gfCNCPoint4[14464] = {X 340.3975, Y 90.3624, Z -5.5000, A 0.000, B 0.000, C 0.000 }
gfCNCPoint4[14465] = {X 344.7798, Y 90.5164, Z -5.5000, A 0.000, B 0.000, C 0.000 }
gfCNCPoint4[14466] = {X 349.1649, Y 90.5297, Z -5.5000, A 0.000, B 0.000, C 0.000 }
gfCNCPoint4[14467] = {X 353.3215, Y 90.4612, Z -5.5000, A 0.000, B 0.000, C 0.000 }
gfCNCPoint4[14468] = {X 357.4730, Y 90.2419, Z -5.5000, A 0.000, B 0.000, C 0.000 }
gfCNCPoint4[14469] = {X 361.6137, Y 89.8721, Z -5.5000, A 0.000, B 0.000, C 0.000 }
gfCNCPoint4[14470] = {X 363.7037, Y 89.5838, Z -5.5000, A 0.000, B 0.000, C 0.000 }
gfCNCPoint4[14471] = {X 365.7746, Y 89.1801, Z -5.5000, A 0.000, B 0.000, C 0.000 }
gfCNCPoint4[14472] = {X 367.8199, Y 88.6622, Z -5.5000, A 0.000, B 0.000, C 0.000 }
gfCNCPoint4[14473] = {X 368.7685, Y 88.3433, Z -5.5000, A 0.000, B 0.000, C 0.000 }
gfCNCPoint4[14474] = {X 369.6754, Y 87.9200, Z -5.5000, A 0.000, B 0.000, C 0.000 }
gfCNCPoint4[14475] = {X 370.5291, Y 87.3978, Z -5.5000, A 0.000, B 0.000, C 0.000 }
gfCNCPoint4[14476] = {X 370.7228, Y 87.1961, Z -5.5000, A 0.000, B 0.000, C 0.000 }
gfCNCPoint4[14477] = {X 370.8227, Y 86.9349, Z -5.5000, A 0.000, B 0.000, C 0.000 }
gfCNCPoint4[14478] = {X 371.0154, Y 85.3870, Z -5.5000, A 0.000, B 0.000, C 0.000 }
gfCNCPoint4[14479] = {X 371.0797, Y 83.8285, Z -5.5000, A 0.000, B 0.000, C 0.000 }
gfCNCPoint4[14480] = {X 371.0803, Y 63.0708, Z -5.5000, A 0.000, B 0.000, C 0.000 }
gfCNCPoint4[14481] = {X 370.9777, Y 63.0587, Z -5.5000, A 0.000, B 0.000, C 0.000 }
gfCNCPoint4[14482] = {X 370.8755, Y 63.0440, Z -5.5000, A 0.000, B 0.000, C 0.000 }
gfCNCPoint4[14483] = {X 369.9381, Y 62.7818, Z -5.5000, A 0.000, B 0.000, C 0.000 }
gfCNCPoint4[14484] = {X 369.0872, Y 62.3091, Z -5.5000, A 0.000, B 0.000, C 0.000 }
gfCNCPoint4[14485] = {X 368.3695, Y 61.6515, Z -5.5000, A 0.000, B 0.000, C 0.000 }
gfCNCPoint4[14486] = {X 367.8242, Y 60.8451, Z -5.5000, A 0.000, B 0.000, C 0.000 }
gfCNCPoint4[14487] = {X 367.4813, Y 59.9342, Z -5.5000, A 0.000, B 0.000, C 0.000 }
gfCNCPoint4[14488] = {X 367.3594, Y 58.9684, Z -5.5000, A 0.000, B 0.000, C 0.000 }
gfCNCPoint4[14489] = {X 367.3593, Y 58.0000, Z -5.5000, A 0.000, B 0.000, C 0.000 }
gfCNCPoint4[14490] = {X 367.4636, Y 57.0743, Z -5.5000, A 0.000, B 0.000, C 0.000 }
gfCNCPoint4[14491] = {X 367.7713, Y 56.1950, Z -5.5000, A 0.000, B 0.000, C 0.000 }
gfCNCPoint4[14492] = {X 368.2669, Y 55.4063, Z -5.5000, A 0.000, B 0.000, C 0.000 }
gfCNCPoint4[14493] = {X 368.9256, Y 54.7476, Z -5.5000, A 0.000, B 0.000, C 0.000 }
gfCNCPoint4[14494] = {X 369.7143, Y 54.2520, Z -5.5000, A 0.000, B 0.000, C 0.000 }
gfCNCPoint4[14495] = {X 370.5936, Y 53.9443, Z -5.5000, A 0.000, B 0.000, C 0.000 }
gfCNCPoint4[14496] = {X 371.5193, Y 53.8400, Z -5.5000, A 0.000, B 0.000, C 0.000 }
gfCNCPoint4[14497] = {X 388.0597, Y 53.8400, Z -5.5000, A 0.000, B 0.000, C 0.000 }
gfCNCPoint4[14498] = {X 388.9854, Y 53.9443, Z -5.5000, A 0.000, B 0.000, C 0.000 }
gfCNCPoint4[14499] = {X 389.8646, Y 54.2520, Z -5.5000, A 0.000, B 0.000, C 0.000 }
gfCNCPoint4[14500] = {X 390.6534, Y 54.7476, Z -5.5000, A 0.000, B 0.000, C 0.000 }
gfCNCPoint4[14501] = {X 391.3121, Y 55.4063, Z -5.5000, A 0.000, B 0.000, C 0.000 }
gfCNCPoint4[14502] = {X 391.8077, Y 56.1950, Z -5.5000, A 0.000, B 0.000, C 0.000 }
gfCNCPoint4[14503] = {X 392.1154, Y 57.0743, Z -5.5000, A 0.000, B 0.000, C 0.000 }
gfCNCPoint4[14504] = {X 392.2197, Y 58.0000, Z -5.5000, A 0.000, B 0.000, C 0.000 }
gfCNCPoint4[14505] = {X 392.2197, Y 58.9342, Z -5.5000, A 0.000, B 0.000, C 0.000 }
gfCNCPoint4[14506] = {X 392.1108, Y 59.8794, Z -5.5000, A 0.000, B 0.000, C 0.000 }
gfCNCPoint4[14507] = {X 391.7901, Y 60.7752, Z -5.5000, A 0.000, B 0.000, C 0.000 }
gfCNCPoint4[14508] = {X 391.2470, Y 61.6084, Z -5.5000, A 0.000, B 0.000, C 0.000 }
gfCNCPoint4[14509] = {X 390.5225, Y 62.2898, Z -5.5000, A 0.000, B 0.000, C 0.000 }
gfCNCPoint4[14510] = {X 389.6577, Y 62.7809, Z -5.5000, A 0.000, B 0.000, C 0.000 }
gfCNCPoint4[14511] = {X 388.7013, Y 63.0540, Z -5.5000, A 0.000, B 0.000, C 0.000 }
gfCNCPoint4[14512] = {X 388.6011, Y 63.0688, Z -5.5000, A 0.000, B 0.000, C 0.000 }
gfCNCPoint4[14513] = {X 388.5005, Y 63.0812, Z -5.5000, A 0.000, B 0.000, C 0.000 }
gfCNCPoint4[14514] = {X 388.4973, Y 84.6154, Z -5.5000, A 0.000, B 0.000, C 0.000 }
gfCNCPoint4[14515] = {X 388.4379, Y 86.2600, Z -5.5000, A 0.000, B 0.000, C 0.000 }
gfCNCPoint4[14516] = {X 388.2353, Y 87.8931, Z -5.5000, A 0.000, B 0.000, C 0.000 }
gfCNCPoint4[14517] = {X 387.8910, Y 89.5023, Z -5.5000, A 0.000, B 0.000, C 0.000 }
gfCNCPoint4[14518] = {X 387.3659, Y 91.0683, Z -5.5000, A 0.000, B 0.000, C 0.000 }
gfCNCPoint4[14519] = {X 386.6264, Y 92.5452, Z -5.5000, A 0.000, B 0.000, C 0.000 }
gfCNCPoint4[14520] = {X 385.6871, Y 93.9038, Z -5.5000, A 0.000, B 0.000, C 0.000 }
gfCNCPoint4[14521] = {X 384.5666, Y 95.1172, Z -5.5000, A 0.000, B 0.000, C 0.000 }
gfCNCPoint4[14522] = {X 383.0651, Y 96.3825, Z -5.5000, A 0.000, B 0.000, C 0.000 }
gfCNCPoint4[14523] = {X 381.4378, Y 97.4811, Z -5.5000, A 0.000, B 0.000, C 0.000 }
gfCNCPoint4[14524] = {X 379.7030, Y 98.4008, Z -5.5000, A 0.000, B 0.000, C 0.000 }
gfCNCPoint4[14525] = {X 377.4420, Y 99.3513, Z -5.5000, A 0.000, B 0.000, C 0.000 }
gfCNCPoint4[14526] = {X 375.1190, Y 100.1379, Z -5.5000, A 0.000, B 0.000, C 0.000 }
gfCNCPoint4[14527] = {X 372.7456, Y 100.7564, Z -5.5000, A 0.000, B 0.000, C 0.000 }
gfCNCPoint4[14528] = {X 368.8428, Y 101.5089, Z -5.5000, A 0.000, B 0.000, C 0.000 }
gfCNCPoint4[14529] = {X 364.9075, Y 102.0681, Z -5.5000, A 0.000, B 0.000, C 0.000 }
gfCNCPoint4[14530] = {X 360.9496, Y 102.4325, Z -5.5000, A 0.000, B 0.000, C 0.000 }
gfCNCPoint4[14531] = {X 357.0957, Y 102.6572, Z -5.5000, A 0.000, B 0.000, C 0.000 }
gfCNCPoint4[14532] = {X 353.2381, Y 102.8025, Z -5.5000, A 0.000, B 0.000, C 0.000 }
gfCNCPoint4[14533] = {X 353.3474, Y 106.8010, Z -5.5000, A 0.000, B 0.000, C 0.000 }
gfCNCPoint4[14534] = {X 353.2359, Y 102.7225, Z -5.5000, A 0.000, B 0.000, C 0.000 }
gfCNCPoint4[14535] = {X 348.1836, Y 102.7923, Z -5.5000, A 0.000, B 0.000, C 0.000 }
gfCNCPoint4[14536] = {X 343.1312, Y 102.7256, Z -5.5000, A 0.000, B 0.000, C 0.000 }
gfCNCPoint4[14537] = {X 338.0825, Y 102.5225, Z -5.5000, A 0.000, B 0.000, C 0.000 }
gfCNCPoint4[14538] = {X 334.1379, Y 102.2462, Z -5.5000, A 0.000, B 0.000, C 0.000 }
gfCNCPoint4[14539] = {X 330.2083, Y 101.8055, Z -5.5000, A 0.000, B 0.000, C 0.000 }
gfCNCPoint4[14540] = {X 326.3005, Y 101.2010, Z -5.5000, A 0.000, B 0.000, C 0.000 }
gfCNCPoint4[14541] = {X 323.4679, Y 100.6003, Z -5.5000, A 0.000, B 0.000, C 0.000 }
gfCNCPoint4[14542] = {X 320.6873, Y 99.7922, Z -5.5000, A 0.000, B 0.000, C 0.000 }
gfCNCPoint4[14543] = {X 317.9740, Y 98.7812, Z -5.5000, A 0.000, B 0.000, C 0.000 }
gfCNCPoint4[14544] = {X 316.4791, Y 98.0919, Z -5.5000, A 0.000, B 0.000, C 0.000 }
gfCNCPoint4[14545] = {X 315.0472, Y 97.2799, Z -5.5000, A 0.000, B 0.000, C 0.000 }
gfCNCPoint4[14546] = {X 313.6882, Y 96.3510, Z -5.5000, A 0.000, B 0.000, C 0.000 }
gfCNCPoint4[14547] = {X 312.4117, Y 95.3116, Z -5.5000, A 0.000, B 0.000, C 0.000 }
gfCNCPoint4[14548] = {X 311.4281, Y 94.3332, Z -5.5000, A 0.000, B 0.000, C 0.000 }
gfCNCPoint4[14549] = {X 310.5674, Y 93.2450, Z -5.5000, A 0.000, B 0.000, C 0.000 }
gfCNCPoint4[14550] = {X 309.8418, Y 92.0625, Z -5.5000, A 0.000, B 0.000, C 0.000 }
gfCNCPoint4[14551] = {X 309.2615, Y 90.8023, Z -5.5000, A 0.000, B 0.000, C 0.000 }
gfCNCPoint4[14552] = {X 308.8346, Y 89.4822, Z -5.5000, A 0.000, B 0.000, C 0.000 }
gfCNCPoint4[14553] = {X 308.4955, Y 87.8792, Z -5.5000, A 0.000, B 0.000, C 0.000 }
gfCNCPoint4[14554] = {X 308.2951, Y 86.2530, Z -5.5000, A 0.000, B 0.000, C 0.000 }
gfCNCPoint4[14555] = {X 308.2350, Y 84.6156, Z -5.5000, A 0.000, B 0.000, C 0.000 }
gfCNCPoint4[14556] = {X 308.2363, Y 62.9982, Z -5.5000, A 0.000, B 0.000, C 0.000 }
gfCNCPoint4[14557] = {X 307.3947, Y 62.8331, Z -5.5000, A 0.000, B 0.000, C 0.000 }
gfCNCPoint4[14558] = {X 306.6061, Y 62.4958, Z -5.5000, A 0.000, B 0.000, C 0.000 }
gfCNCPoint4[14559] = {X 305.9055, Y 62.0011, Z -5.5000, A 0.000, B 0.000, C 0.000 }
gfCNCPoint4[14560] = {X 305.3238, Y 61.3708, Z -5.5000, A 0.000, B 0.000, C 0.000 }
gfCNCPoint4[14561] = {X 304.8867, Y 60.6329, Z -5.5000, A 0.000, B 0.000, C 0.000 }
gfCNCPoint4[14562] = {X 304.6136, Y 59.8199, Z -5.5000, A 0.000, B 0.000, C 0.000 }
gfCNCPoint4[14563] = {X 304.5164, Y 58.9678, Z -5.5000, A 0.000, B 0.000, C 0.000 }
gfCNCPoint4[14564] = {X 304.5162, Y 58.0000, Z -5.5000, A 0.000, B 0.000, C 0.000 }
gfCNCPoint4[14565] = {X 304.6185, Y 57.0921, Z -5.5000, A 0.000, B 0.000, C 0.000 }
gfCNCPoint4[14566] = {X 304.9203, Y 56.2298, Z -5.5000, A 0.000, B 0.000, C 0.000 }
gfCNCPoint4[14567] = {X 305.4064, Y 55.4562, Z -5.5000, A 0.000, B 0.000, C 0.000 }
gfCNCPoint4[14568] = {X 306.0524, Y 54.8101, Z -5.5000, A 0.000, B 0.000, C 0.000 }
gfCNCPoint4[14569] = {X 306.8260, Y 54.3240, Z -5.5000, A 0.000, B 0.000, C 0.000 }
gfCNCPoint4[14570] = {X 307.6883, Y 54.0223, Z -5.5000, A 0.000, B 0.000, C 0.000 }
gfCNCPoint4[14571] = {X 308.5962, Y 53.9200, Z -5.5000, A 0.000, B 0.000, C 0.000 }
gfCNCPoint4[14572] = {X 324.3107, Y 53.9200, Z -5.5000, A 0.000, B 0.000, C 0.000 }
gfCNCPoint4[14573] = {X 325.2186, Y 54.0223, Z -5.5000, A 0.000, B 0.000, C 0.000 }
gfCNCPoint4[14574] = {X 326.0809, Y 54.3240, Z -5.5000, A 0.000, B 0.000, C 0.000 }
gfCNCPoint4[14575] = {X 326.8545, Y 54.8101, Z -5.5000, A 0.000, B 0.000, C 0.000 }
gfCNCPoint4[14576] = {X 327.5006, Y 55.4562, Z -5.5000, A 0.000, B 0.000, C 0.000 }
gfCNCPoint4[14577] = {X 327.9866, Y 56.2298, Z -5.5000, A 0.000, B 0.000, C 0.000 }
gfCNCPoint4[14578] = {X 328.2884, Y 57.0921, Z -5.5000, A 0.000, B 0.000, C 0.000 }
gfCNCPoint4[14579] = {X 328.3907, Y 58.0000, Z -5.5000, A 0.000, B 0.000, C 0.000 }
gfCNCPoint4[14580] = {X 328.3907, Y 58.9345, Z -5.5000, A 0.000, B 0.000, C 0.000 }
gfCNCPoint4[14581] = {X 328.2957, Y 59.7914, Z -5.5000, A 0.000, B 0.000, C 0.000 }
gfCNCPoint4[14582] = {X 328.0243, Y 60.6097, Z -5.5000, A 0.000, B 0.000, C 0.000 }
gfCNCPoint4[14583] = {X 327.5886, Y 61.3536, Z -5.5000, A 0.000, B 0.000, C 0.000 }
gfCNCPoint4[14584] = {X 327.0075, Y 61.9905, Z -5.5000, A 0.000, B 0.000, C 0.000 }
gfCNCPoint4[14585] = {X 326.3065, Y 62.4924, Z -5.5000, A 0.000, B 0.000, C 0.000 }
gfCNCPoint4[14586] = {X 325.5164, Y 62.8374, Z -5.5000, A 0.000, B 0.000, C 0.000 }
gfCNCPoint4[14587] = {X 324.6718, Y 63.0103, Z -5.5000, A 0.000, B 0.000, C 0.000 }
gfCNCPoint4[14588] = {X 324.6736, Y 83.2308, Z -5.5000, A 0.000, B 0.000, C 0.000 }
gfCNCPoint4[14589] = {X 324.6871, Y 84.6156, Z -5.5000, A 0.000, B 0.000, C 0.000 }
gfCNCPoint4[14590] = {X 324.7690, Y 85.9011, Z -5.5000, A 0.000, B 0.000, C 0.000 }
gfCNCPoint4[14591] = {X 325.0037, Y 87.1677, Z -5.5000, A 0.000, B 0.000, C 0.000 }
gfCNCPoint4[14592] = {X 325.2950, Y 87.5003, Z -5.5000, A 0.000, B 0.000, C 0.000 }
gfCNCPoint4[14593] = {X 325.6599, Y 87.7499, Z -5.5000, A 0.000, B 0.000, C 0.000 }
gfCNCPoint4[14594] = {X 326.1137, Y 88.0066, Z -5.5000, A 0.000, B 0.000, C 0.000 }
gfCNCPoint4[14595] = {X 327.5791, Y 88.6152, Z -5.5000, A 0.000, B 0.000, C 0.000 }
gfCNCPoint4[14596] = {X 329.1025, Y 89.0594, Z -5.5000, A 0.000, B 0.000, C 0.000 }
gfCNCPoint4[14597] = {X 331.3881, Y 89.5353, Z -5.5000, A 0.000, B 0.000, C 0.000 }
gfCNCPoint4[14598] = {X 333.6944, Y 89.8982, Z -5.5000, A 0.000, B 0.000, C 0.000 }
gfCNCPoint4[14599] = {X 336.0157, Y 90.1475, Z -5.5000, A 0.000, B 0.000, C 0.000 }
gfCNCPoint4[14600] = {X 340.3934, Y 90.4423, Z -5.5000, A 0.000, B 0.000, C 0.000 }
gfCNCPoint4[14601] = {X 344.7783, Y 90.5964, Z -5.5000, A 0.000, B 0.000, C 0.000 }
gfCNCPoint4[14602] = {X 349.1659, Y 90.6096, Z -5.5000, A 0.000, B 0.000, C 0.000 }
gfCNCPoint4[14603] = {X 353.3251, Y 90.5411, Z -5.5000, A 0.000, B 0.000, C 0.000 }
gfCNCPoint4[14604] = {X 357.4791, Y 90.3217, Z -5.5000, A 0.000, B 0.000, C 0.000 }
gfCNCPoint4[14605] = {X 361.6223, Y 89.9516, Z -5.5000, A 0.000, B 0.000, C 0.000 }
gfCNCPoint4[14606] = {X 363.7168, Y 89.6627, Z -5.5000, A 0.000, B 0.000, C 0.000 }
gfCNCPoint4[14607] = {X 365.7920, Y 89.2582, Z -5.5000, A 0.000, B 0.000, C 0.000 }
gfCNCPoint4[14608] = {X 367.8417, Y 88.7392, Z -5.5000, A 0.000, B 0.000, C 0.000 }
gfCNCPoint4[14609] = {X 368.7986, Y 88.4174, Z -5.5000, A 0.000, B 0.000, C 0.000 }
gfCNCPoint4[14610] = {X 369.7134, Y 87.9904, Z -5.5000, A 0.000, B 0.000, C 0.000 }
gfCNCPoint4[14611] = {X 370.5746, Y 87.4635, Z -5.5000, A 0.000, B 0.000, C 0.000 }
gfCNCPoint4[14612] = {X 370.7904, Y 87.2390, Z -5.5000, A 0.000, B 0.000, C 0.000 }
gfCNCPoint4[14613] = {X 370.9016, Y 86.9481, Z -5.5000, A 0.000, B 0.000, C 0.000 }
gfCNCPoint4[14614] = {X 371.0952, Y 85.3936, Z -5.5000, A 0.000, B 0.000, C 0.000 }
gfCNCPoint4[14615] = {X 371.1597, Y 83.8285, Z -5.5000, A 0.000, B 0.000, C 0.000 }
gfCNCPoint4[14616] = {X 371.1603, Y 62.9982, Z -5.5000, A 0.000, B 0.000, C 0.000 }
gfCNCPoint4[14617] = {X 371.0238, Y 62.9839, Z -5.5000, A 0.000, B 0.000, C 0.000 }
gfCNCPoint4[14618] = {X 370.8879, Y 62.9649, Z -5.5000, A 0.000, B 0.000, C 0.000 }
gfCNCPoint4[14619] = {X 369.9685, Y 62.7078, Z -5.5000, A 0.000, B 0.000, C 0.000 }
gfCNCPoint4[14620] = {X 369.1340, Y 62.2442, Z -5.5000, A 0.000, B 0.000, C 0.000 }
gfCNCPoint4[14621] = {X 368.4301, Y 61.5992, Z -5.5000, A 0.000, B 0.000, C 0.000 }
gfCNCPoint4[14622] = {X 367.8953, Y 60.8084, Z -5.5000, A 0.000, B 0.000, C 0.000 }
gfCNCPoint4[14623] = {X 367.5589, Y 59.9149, Z -5.5000, A 0.000, B 0.000, C 0.000 }
gfCNCPoint4[14624] = {X 367.4394, Y 58.9678, Z -5.5000, A 0.000, B 0.000, C 0.000 }
gfCNCPoint4[14625] = {X 367.4393, Y 58.0000, Z -5.5000, A 0.000, B 0.000, C 0.000 }
gfCNCPoint4[14626] = {X 367.5416, Y 57.0921, Z -5.5000, A 0.000, B 0.000, C 0.000 }
gfCNCPoint4[14627] = {X 367.8433, Y 56.2298, Z -5.5000, A 0.000, B 0.000, C 0.000 }
gfCNCPoint4[14628] = {X 368.3294, Y 55.4562, Z -5.5000, A 0.000, B 0.000, C 0.000 }
gfCNCPoint4[14629] = {X 368.9754, Y 54.8101, Z -5.5000, A 0.000, B 0.000, C 0.000 }
gfCNCPoint4[14630] = {X 369.7490, Y 54.3240, Z -5.5000, A 0.000, B 0.000, C 0.000 }
gfCNCPoint4[14631] = {X 370.6114, Y 54.0223, Z -5.5000, A 0.000, B 0.000, C 0.000 }
gfCNCPoint4[14632] = {X 371.5193, Y 53.9200, Z -5.5000, A 0.000, B 0.000, C 0.000 }
gfCNCPoint4[14633] = {X 388.0597, Y 53.9200, Z -5.5000, A 0.000, B 0.000, C 0.000 }
gfCNCPoint4[14634] = {X 388.9676, Y 54.0223, Z -5.5000, A 0.000, B 0.000, C 0.000 }
gfCNCPoint4[14635] = {X 389.8299, Y 54.3240, Z -5.5000, A 0.000, B 0.000, C 0.000 }
gfCNCPoint4[14636] = {X 390.6035, Y 54.8101, Z -5.5000, A 0.000, B 0.000, C 0.000 }
gfCNCPoint4[14637] = {X 391.2496, Y 55.4562, Z -5.5000, A 0.000, B 0.000, C 0.000 }
gfCNCPoint4[14638] = {X 391.7356, Y 56.2298, Z -5.5000, A 0.000, B 0.000, C 0.000 }
gfCNCPoint4[14639] = {X 392.0374, Y 57.0921, Z -5.5000, A 0.000, B 0.000, C 0.000 }
gfCNCPoint4[14640] = {X 392.1397, Y 58.0000, Z -5.5000, A 0.000, B 0.000, C 0.000 }
gfCNCPoint4[14641] = {X 392.1397, Y 58.9342, Z -5.5000, A 0.000, B 0.000, C 0.000 }
gfCNCPoint4[14642] = {X 392.0329, Y 59.8612, Z -5.5000, A 0.000, B 0.000, C 0.000 }
gfCNCPoint4[14643] = {X 391.7183, Y 60.7398, Z -5.5000, A 0.000, B 0.000, C 0.000 }
gfCNCPoint4[14644] = {X 391.1856, Y 61.5570, Z -5.5000, A 0.000, B 0.000, C 0.000 }
gfCNCPoint4[14645] = {X 390.4750, Y 62.2254, Z -5.5000, A 0.000, B 0.000, C 0.000 }
gfCNCPoint4[14646] = {X 389.6267, Y 62.7072, Z -5.5000, A 0.000, B 0.000, C 0.000 }
gfCNCPoint4[14647] = {X 388.6887, Y 62.9750, Z -5.5000, A 0.000, B 0.000, C 0.000 }
gfCNCPoint4[14648] = {X 388.5554, Y 62.9941, Z -5.5000, A 0.000, B 0.000, C 0.000 }
gfCNCPoint4[14649] = {X 388.4216, Y 63.0089, Z -5.5000, A 0.000, B 0.000, C 0.000 }
gfCNCPoint4[14650] = {X 388.4193, Y 63.1547, Z -5.5000, A 0.000, B 0.000, C 0.000 }
gfCNCPoint4[14651] = {X 388.4173, Y 84.6157, Z -5.5000, A 0.000, B 0.000, C 0.000 }
gfCNCPoint4[14652] = {X 388.3582, Y 86.2534, Z -5.5000, A 0.000, B 0.000, C 0.000 }
gfCNCPoint4[14653] = {X 388.1564, Y 87.8797, Z -5.5000, A 0.000, B 0.000, C 0.000 }
gfCNCPoint4[14654] = {X 387.8135, Y 89.4823, Z -5.5000, A 0.000, B 0.000, C 0.000 }
gfCNCPoint4[14655] = {X 387.2920, Y 91.0376, Z -5.5000, A 0.000, B 0.000, C 0.000 }
gfCNCPoint4[14656] = {X 386.5576, Y 92.5044, Z -5.5000, A 0.000, B 0.000, C 0.000 }
gfCNCPoint4[14657] = {X 385.6247, Y 93.8538, Z -5.5000, A 0.000, B 0.000, C 0.000 }
gfCNCPoint4[14658] = {X 384.5117, Y 95.0589, Z -5.5000, A 0.000, B 0.000, C 0.000 }
gfCNCPoint4[14659] = {X 383.0168, Y 96.3187, Z -5.5000, A 0.000, B 0.000, C 0.000 }
gfCNCPoint4[14660] = {X 381.3966, Y 97.4125, Z -5.5000, A 0.000, B 0.000, C 0.000 }
gfCNCPoint4[14661] = {X 379.6693, Y 98.3282, Z -5.5000, A 0.000, B 0.000, C 0.000 }
gfCNCPoint4[14662] = {X 377.4137, Y 99.2765, Z -5.5000, A 0.000, B 0.000, C 0.000 }
gfCNCPoint4[14663] = {X 375.0960, Y 100.0612, Z -5.5000, A 0.000, B 0.000, C 0.000 }
gfCNCPoint4[14664] = {X 372.7282, Y 100.6783, Z -5.5000, A 0.000, B 0.000, C 0.000 }
gfCNCPoint4[14665] = {X 368.8293, Y 101.4301, Z -5.5000, A 0.000, B 0.000, C 0.000 }
gfCNCPoint4[14666] = {X 364.8981, Y 101.9887, Z -5.5000, A 0.000, B 0.000, C 0.000 }
gfCNCPoint4[14667] = {X 360.9441, Y 102.3527, Z -5.5000, A 0.000, B 0.000, C 0.000 }
gfCNCPoint4[14668] = {X 357.0919, Y 102.5773, Z -5.5000, A 0.000, B 0.000, C 0.000 }
gfCNCPoint4[14669] = {X 353.2359, Y 102.7225, Z -5.5000, A 0.000, B 0.000, C 0.000 }
gfCNCPoint4[14670] = {X 353.3452, Y 106.7210, Z -5.5000, A 0.000, B 0.000, C 0.000 }
gfCNCPoint4[14671] = {X 353.2337, Y 102.6425, Z -5.5000, A 0.000, B 0.000, C 0.000 }
gfCNCPoint4[14672] = {X 348.1835, Y 102.7123, Z -5.5000, A 0.000, B 0.000, C 0.000 }
gfCNCPoint4[14673] = {X 343.1332, Y 102.6456, Z -5.5000, A 0.000, B 0.000, C 0.000 }
gfCNCPoint4[14674] = {X 338.0866, Y 102.4426, Z -5.5000, A 0.000, B 0.000, C 0.000 }
gfCNCPoint4[14675] = {X 334.1453, Y 102.1666, Z -5.5000, A 0.000, B 0.000, C 0.000 }
gfCNCPoint4[14676] = {X 330.2189, Y 101.7262, Z -5.5000, A 0.000, B 0.000, C 0.000 }
gfCNCPoint4[14677] = {X 326.3144, Y 101.1222, Z -5.5000, A 0.000, B 0.000, C 0.000 }
gfCNCPoint4[14678] = {X 323.4875, Y 100.5227, Z -5.5000, A 0.000, B 0.000, C 0.000 }
gfCNCPoint4[14679] = {X 320.7125, Y 99.7163, Z -5.5000, A 0.000, B 0.000, C 0.000 }
gfCNCPoint4[14680] = {X 318.0046, Y 98.7073, Z -5.5000, A 0.000, B 0.000, C 0.000 }
gfCNCPoint4[14681] = {X 316.5158, Y 98.0207, Z -5.5000, A 0.000, B 0.000, C 0.000 }
gfCNCPoint4[14682] = {X 315.0896, Y 97.2121, Z -5.5000, A 0.000, B 0.000, C 0.000 }
gfCNCPoint4[14683] = {X 313.7361, Y 96.2869, Z -5.5000, A 0.000, B 0.000, C 0.000 }
gfCNCPoint4[14684] = {X 312.4647, Y 95.2517, Z -5.5000, A 0.000, B 0.000, C 0.000 }
gfCNCPoint4[14685] = {X 311.4878, Y 94.2800, Z -5.5000, A 0.000, B 0.000, C 0.000 }
gfCNCPoint4[14686] = {X 310.6330, Y 93.1992, Z -5.5000, A 0.000, B 0.000, C 0.000 }
gfCNCPoint4[14687] = {X 309.9124, Y 92.0248, Z -5.5000, A 0.000, B 0.000, C 0.000 }
gfCNCPoint4[14688] = {X 309.3360, Y 90.7732, Z -5.5000, A 0.000, B 0.000, C 0.000 }
gfCNCPoint4[14689] = {X 308.9121, Y 89.4621, Z -5.5000, A 0.000, B 0.000, C 0.000 }
gfCNCPoint4[14690] = {X 308.5744, Y 87.8658, Z -5.5000, A 0.000, B 0.000, C 0.000 }
gfCNCPoint4[14691] = {X 308.3749, Y 86.2464, Z -5.5000, A 0.000, B 0.000, C 0.000 }
gfCNCPoint4[14692] = {X 308.3150, Y 84.6159, Z -5.5000, A 0.000, B 0.000, C 0.000 }
gfCNCPoint4[14693] = {X 308.3163, Y 62.9243, Z -5.5000, A 0.000, B 0.000, C 0.000 }
gfCNCPoint4[14694] = {X 307.4738, Y 62.7734, Z -5.5000, A 0.000, B 0.000, C 0.000 }
gfCNCPoint4[14695] = {X 306.6826, Y 62.4466, Z -5.5000, A 0.000, B 0.000, C 0.000 }
gfCNCPoint4[14696] = {X 305.9791, Y 61.9591, Z -5.5000, A 0.000, B 0.000, C 0.000 }
gfCNCPoint4[14697] = {X 305.3955, Y 61.3330, Z -5.5000, A 0.000, B 0.000, C 0.000 }
gfCNCPoint4[14698] = {X 304.9583, Y 60.5971, Z -5.5000, A 0.000, B 0.000, C 0.000 }
gfCNCPoint4[14699] = {X 304.6878, Y 59.7851, Z -5.5000, A 0.000, B 0.000, C 0.000 }
gfCNCPoint4[14700] = {X 304.5962, Y 58.9341, Z -5.5000, A 0.000, B 0.000, C 0.000 }
gfCNCPoint4[14701] = {X 304.5962, Y 58.0000, Z -5.5000, A 0.000, B 0.000, C 0.000 }
gfCNCPoint4[14702] = {X 304.6965, Y 57.1099, Z -5.5000, A 0.000, B 0.000, C 0.000 }
gfCNCPoint4[14703] = {X 304.9923, Y 56.2645, Z -5.5000, A 0.000, B 0.000, C 0.000 }
gfCNCPoint4[14704] = {X 305.4689, Y 55.5060, Z -5.5000, A 0.000, B 0.000, C 0.000 }
gfCNCPoint4[14705] = {X 306.1023, Y 54.8727, Z -5.5000, A 0.000, B 0.000, C 0.000 }
gfCNCPoint4[14706] = {X 306.8607, Y 54.3961, Z -5.5000, A 0.000, B 0.000, C 0.000 }
gfCNCPoint4[14707] = {X 307.7061, Y 54.1003, Z -5.5000, A 0.000, B 0.000, C 0.000 }
gfCNCPoint4[14708] = {X 308.5962, Y 54.0000, Z -5.5000, A 0.000, B 0.000, C 0.000 }
gfCNCPoint4[14709] = {X 324.3107, Y 54.0000, Z -5.5000, A 0.000, B 0.000, C 0.000 }
gfCNCPoint4[14710] = {X 325.2008, Y 54.1003, Z -5.5000, A 0.000, B 0.000, C 0.000 }
gfCNCPoint4[14711] = {X 326.0462, Y 54.3961, Z -5.5000, A 0.000, B 0.000, C 0.000 }
gfCNCPoint4[14712] = {X 326.8046, Y 54.8727, Z -5.5000, A 0.000, B 0.000, C 0.000 }
gfCNCPoint4[14713] = {X 327.4380, Y 55.5060, Z -5.5000, A 0.000, B 0.000, C 0.000 }
gfCNCPoint4[14714] = {X 327.9146, Y 56.2645, Z -5.5000, A 0.000, B 0.000, C 0.000 }
gfCNCPoint4[14715] = {X 328.2104, Y 57.1099, Z -5.5000, A 0.000, B 0.000, C 0.000 }
gfCNCPoint4[14716] = {X 328.3107, Y 58.0000, Z -5.5000, A 0.000, B 0.000, C 0.000 }
gfCNCPoint4[14717] = {X 328.3107, Y 58.9341, Z -5.5000, A 0.000, B 0.000, C 0.000 }
gfCNCPoint4[14718] = {X 328.2153, Y 59.7844, Z -5.5000, A 0.000, B 0.000, C 0.000 }
gfCNCPoint4[14719] = {X 327.9429, Y 60.5956, Z -5.5000, A 0.000, B 0.000, C 0.000 }
gfCNCPoint4[14720] = {X 327.5056, Y 61.3311, Z -5.5000, A 0.000, B 0.000, C 0.000 }
gfCNCPoint4[14721] = {X 326.9232, Y 61.9580, Z -5.5000, A 0.000, B 0.000, C 0.000 }
gfCNCPoint4[14722] = {X 326.2218, Y 62.4481, Z -5.5000, A 0.000, B 0.000, C 0.000 }
gfCNCPoint4[14723] = {X 325.4328, Y 62.7794, Z -5.5000, A 0.000, B 0.000, C 0.000 }
gfCNCPoint4[14724] = {X 324.5918, Y 62.9370, Z -5.5000, A 0.000, B 0.000, C 0.000 }
gfCNCPoint4[14725] = {X 324.5936, Y 83.2313, Z -5.5000, A 0.000, B 0.000, C 0.000 }
gfCNCPoint4[14726] = {X 324.6071, Y 84.6159, Z -5.5000, A 0.000, B 0.000, C 0.000 }
gfCNCPoint4[14727] = {X 324.6905, Y 85.9179, Z -5.5000, A 0.000, B 0.000, C 0.000 }
gfCNCPoint4[14728] = {X 324.9294, Y 87.2005, Z -5.5000, A 0.000, B 0.000, C 0.000 }
gfCNCPoint4[14729] = {X 325.2359, Y 87.5548, Z -5.5000, A 0.000, B 0.000, C 0.000 }
gfCNCPoint4[14730] = {X 325.6219, Y 87.8203, Z -5.5000, A 0.000, B 0.000, C 0.000 }
gfCNCPoint4[14731] = {X 326.0766, Y 88.0775, Z -5.5000, A 0.000, B 0.000, C 0.000 }
gfCNCPoint4[14732] = {X 327.5513, Y 88.6903, Z -5.5000, A 0.000, B 0.000, C 0.000 }
gfCNCPoint4[14733] = {X 329.0843, Y 89.1373, Z -5.5000, A 0.000, B 0.000, C 0.000 }
gfCNCPoint4[14734] = {X 331.3738, Y 89.6140, Z -5.5000, A 0.000, B 0.000, C 0.000 }
gfCNCPoint4[14735] = {X 333.6840, Y 89.9775, Z -5.5000, A 0.000, B 0.000, C 0.000 }
gfCNCPoint4[14736] = {X 336.0092, Y 90.2272, Z -5.5000, A 0.000, B 0.000, C 0.000 }
gfCNCPoint4[14737] = {X 340.3892, Y 90.5221, Z -5.5000, A 0.000, B 0.000, C 0.000 }
gfCNCPoint4[14738] = {X 344.7764, Y 90.6763, Z -5.5000, A 0.000, B 0.000, C 0.000 }
gfCNCPoint4[14739] = {X 349.1664, Y 90.6896, Z -5.5000, A 0.000, B 0.000, C 0.000 }
gfCNCPoint4[14740] = {X 353.3283, Y 90.6211, Z -5.5000, A 0.000, B 0.000, C 0.000 }
gfCNCPoint4[14741] = {X 357.4851, Y 90.4015, Z -5.5000, A 0.000, B 0.000, C 0.000 }
gfCNCPoint4[14742] = {X 361.6311, Y 90.0311, Z -5.5000, A 0.000, B 0.000, C 0.000 }
gfCNCPoint4[14743] = {X 363.7299, Y 89.7416, Z -5.5000, A 0.000, B 0.000, C 0.000 }
gfCNCPoint4[14744] = {X 365.8095, Y 89.3362, Z -5.5000, A 0.000, B 0.000, C 0.000 }
gfCNCPoint4[14745] = {X 367.8634, Y 88.8162, Z -5.5000, A 0.000, B 0.000, C 0.000 }
gfCNCPoint4[14746] = {X 368.8287, Y 88.4916, Z -5.5000, A 0.000, B 0.000, C 0.000 }
gfCNCPoint4[14747] = {X 369.7514, Y 88.0608, Z -5.5000, A 0.000, B 0.000, C 0.000 }
gfCNCPoint4[14748] = {X 370.6201, Y 87.5293, Z -5.5000, A 0.000, B 0.000, C 0.000 }
gfCNCPoint4[14749] = {X 370.8579, Y 87.2818, Z -5.5000, A 0.000, B 0.000, C 0.000 }
gfCNCPoint4[14750] = {X 370.9805, Y 86.9612, Z -5.5000, A 0.000, B 0.000, C 0.000 }
gfCNCPoint4[14751] = {X 371.1749, Y 85.4002, Z -5.5000, A 0.000, B 0.000, C 0.000 }
gfCNCPoint4[14752] = {X 371.2397, Y 83.8285, Z -5.5000, A 0.000, B 0.000, C 0.000 }
gfCNCPoint4[14753] = {X 371.2384, Y 63.0394, Z -5.5000, A 0.000, B 0.000, C 0.000 }
gfCNCPoint4[14754] = {X 371.2440, Y 62.9246, Z -5.5000, A 0.000, B 0.000, C 0.000 }
gfCNCPoint4[14755] = {X 371.0717, Y 62.9090, Z -5.5000, A 0.000, B 0.000, C 0.000 }
gfCNCPoint4[14756] = {X 370.9003, Y 62.8859, Z -5.5000, A 0.000, B 0.000, C 0.000 }
gfCNCPoint4[14757] = {X 369.9938, Y 62.6318, Z -5.5000, A 0.000, B 0.000, C 0.000 }
gfCNCPoint4[14758] = {X 369.1718, Y 62.1728, Z -5.5000, A 0.000, B 0.000, C 0.000 }
gfCNCPoint4[14759] = {X 368.4799, Y 61.5344, Z -5.5000, A 0.000, B 0.000, C 0.000 }
gfCNCPoint4[14760] = {X 367.9563, Y 60.7520, Z -5.5000, A 0.000, B 0.000, C 0.000 }
gfCNCPoint4[14761] = {X 367.6301, Y 59.8689, Z -5.5000, A 0.000, B 0.000, C 0.000 }
gfCNCPoint4[14762] = {X 367.5193, Y 58.9341, Z -5.5000, A 0.000, B 0.000, C 0.000 }
gfCNCPoint4[14763] = {X 367.5193, Y 58.0000, Z -5.5000, A 0.000, B 0.000, C 0.000 }
gfCNCPoint4[14764] = {X 367.6196, Y 57.1099, Z -5.5000, A 0.000, B 0.000, C 0.000 }
gfCNCPoint4[14765] = {X 367.9154, Y 56.2645, Z -5.5000, A 0.000, B 0.000, C 0.000 }
gfCNCPoint4[14766] = {X 368.3920, Y 55.5060, Z -5.5000, A 0.000, B 0.000, C 0.000 }
gfCNCPoint4[14767] = {X 369.0253, Y 54.8727, Z -5.5000, A 0.000, B 0.000, C 0.000 }
gfCNCPoint4[14768] = {X 369.7837, Y 54.3961, Z -5.5000, A 0.000, B 0.000, C 0.000 }
gfCNCPoint4[14769] = {X 370.6292, Y 54.1003, Z -5.5000, A 0.000, B 0.000, C 0.000 }
gfCNCPoint4[14770] = {X 371.5193, Y 54.0000, Z -5.5000, A 0.000, B 0.000, C 0.000 }
gfCNCPoint4[14771] = {X 388.0597, Y 54.0000, Z -5.5000, A 0.000, B 0.000, C 0.000 }
gfCNCPoint4[14772] = {X 388.9498, Y 54.1003, Z -5.5000, A 0.000, B 0.000, C 0.000 }
gfCNCPoint4[14773] = {X 389.7952, Y 54.3961, Z -5.5000, A 0.000, B 0.000, C 0.000 }
gfCNCPoint4[14774] = {X 390.5536, Y 54.8727, Z -5.5000, A 0.000, B 0.000, C 0.000 }
gfCNCPoint4[14775] = {X 391.1870, Y 55.5060, Z -5.5000, A 0.000, B 0.000, C 0.000 }
gfCNCPoint4[14776] = {X 391.6636, Y 56.2645, Z -5.5000, A 0.000, B 0.000, C 0.000 }
gfCNCPoint4[14777] = {X 391.9594, Y 57.1099, Z -5.5000, A 0.000, B 0.000, C 0.000 }
gfCNCPoint4[14778] = {X 392.0597, Y 58.0000, Z -5.5000, A 0.000, B 0.000, C 0.000 }
gfCNCPoint4[14779] = {X 392.0595, Y 58.9671, Z -5.5000, A 0.000, B 0.000, C 0.000 }
gfCNCPoint4[14780] = {X 391.9513, Y 59.8591, Z -5.5000, A 0.000, B 0.000, C 0.000 }
gfCNCPoint4[14781] = {X 391.6466, Y 60.7044, Z -5.5000, A 0.000, B 0.000, C 0.000 }
gfCNCPoint4[14782] = {X 391.1243, Y 61.5057, Z -5.5000, A 0.000, B 0.000, C 0.000 }
gfCNCPoint4[14783] = {X 390.4275, Y 62.1611, Z -5.5000, A 0.000, B 0.000, C 0.000 }
gfCNCPoint4[14784] = {X 389.5958, Y 62.6334, Z -5.5000, A 0.000, B 0.000, C 0.000 }
gfCNCPoint4[14785] = {X 388.6760, Y 62.8960, Z -5.5000, A 0.000, B 0.000, C 0.000 }
gfCNCPoint4[14786] = {X 388.5098, Y 62.9191, Z -5.5000, A 0.000, B 0.000, C 0.000 }
gfCNCPoint4[14787] = {X 388.3427, Y 62.9353, Z -5.5000, A 0.000, B 0.000, C 0.000 }
gfCNCPoint4[14788] = {X 388.3393, Y 63.1540, Z -5.5000, A 0.000, B 0.000, C 0.000 }
gfCNCPoint4[14789] = {X 388.3393, Y 83.9236, Z -5.5000, A 0.000, B 0.000, C 0.000 }
gfCNCPoint4[14790] = {X 388.3373, Y 84.6159, Z -5.5000, A 0.000, B 0.000, C 0.000 }
gfCNCPoint4[14791] = {X 388.2784, Y 86.2468, Z -5.5000, A 0.000, B 0.000, C 0.000 }
gfCNCPoint4[14792] = {X 388.0775, Y 87.8663, Z -5.5000, A 0.000, B 0.000, C 0.000 }
gfCNCPoint4[14793] = {X 387.7361, Y 89.4621, Z -5.5000, A 0.000, B 0.000, C 0.000 }
gfCNCPoint4[14794] = {X 387.2182, Y 91.0068, Z -5.5000, A 0.000, B 0.000, C 0.000 }
gfCNCPoint4[14795] = {X 386.4888, Y 92.4636, Z -5.5000, A 0.000, B 0.000, C 0.000 }
gfCNCPoint4[14796] = {X 385.5622, Y 93.8037, Z -5.5000, A 0.000, B 0.000, C 0.000 }
gfCNCPoint4[14797] = {X 384.4569, Y 95.0007, Z -5.5000, A 0.000, B 0.000, C 0.000 }
gfCNCPoint4[14798] = {X 382.9685, Y 96.2549, Z -5.5000, A 0.000, B 0.000, C 0.000 }
gfCNCPoint4[14799] = {X 381.3553, Y 97.3440, Z -5.5000, A 0.000, B 0.000, C 0.000 }
gfCNCPoint4[14800] = {X 379.6357, Y 98.2556, Z -5.5000, A 0.000, B 0.000, C 0.000 }
gfCNCPoint4[14801] = {X 377.3853, Y 99.2017, Z -5.5000, A 0.000, B 0.000, C 0.000 }
gfCNCPoint4[14802] = {X 375.0731, Y 99.9846, Z -5.5000, A 0.000, B 0.000, C 0.000 }
gfCNCPoint4[14803] = {X 372.7108, Y 100.6002, Z -5.5000, A 0.000, B 0.000, C 0.000 }
gfCNCPoint4[14804] = {X 368.8159, Y 101.3512, Z -5.5000, A 0.000, B 0.000, C 0.000 }
gfCNCPoint4[14805] = {X 364.8886, Y 101.9092, Z -5.5000, A 0.000, B 0.000, C 0.000 }
gfCNCPoint4[14806] = {X 360.9386, Y 102.2729, Z -5.5000, A 0.000, B 0.000, C 0.000 }
gfCNCPoint4[14807] = {X 357.0881, Y 102.4974, Z -5.5000, A 0.000, B 0.000, C 0.000 }
gfCNCPoint4[14808] = {X 353.2337, Y 102.6425, Z -5.5000, A 0.000, B 0.000, C 0.000 }
gfCNCPoint4[14809] = {X 353.3452, Y 106.7210, Z -5.5000, A 0.000, B 0.000, C 0.000 }
gfCNCPoint4[14810] = {X 353.3452, Y 106.7210, Z -2.5000, A 0.000, B 0.000, C 0.000 }
gfCNCPoint4[14811] = {X 353.3452, Y 106.7210, Z 11.0000, A 0.000, B 0.000, C 0.000 }
gfCNCPoint4[14812] = {X 411.5987, Y 79.5925, Z 11.0000, A 0.000, B 0.000, C 0.000 }
gfCNCPoint4[14813] = {X 411.5987, Y 79.5925, Z -2.5000, A 0.000, B 0.000, C 0.000 }
gfCNCPoint4[14814] = {X 411.5987, Y 79.5925, Z -5.5000, A 0.000, B 0.000, C 0.000 }
gfCNCPoint4[14815] = {X 413.7990, Y 83.0284, Z -5.5000, A 0.000, B 0.000, C 0.000 }
gfCNCPoint4[14816] = {X 428.0542, Y 73.8996, Z -5.5000, A 0.000, B 0.000, C 0.000 }
gfCNCPoint4[14817] = {X 403.7555, Y 64.3662, Z -5.5000, A 0.000, B 0.000, C 0.000 }
gfCNCPoint4[14818] = {X 402.0596, Y 63.8047, Z -5.5000, A 0.000, B 0.000, C 0.000 }
gfCNCPoint4[14819] = {X 400.3123, Y 63.4325, Z -5.5000, A 0.000, B 0.000, C 0.000 }
gfCNCPoint4[14820] = {X 398.5348, Y 63.2540, Z -5.5000, A 0.000, B 0.000, C 0.000 }
gfCNCPoint4[14821] = {X 397.5823, Y 63.1425, Z -5.5000, A 0.000, B 0.000, C 0.000 }
gfCNCPoint4[14822] = {X 396.6778, Y 62.8236, Z -5.5000, A 0.000, B 0.000, C 0.000 }
gfCNCPoint4[14823] = {X 395.8660, Y 62.3130, Z -5.5000, A 0.000, B 0.000, C 0.000 }
gfCNCPoint4[14824] = {X 395.1869, Y 61.6359, Z -5.5000, A 0.000, B 0.000, C 0.000 }
gfCNCPoint4[14825] = {X 394.6739, Y 60.8256, Z -5.5000, A 0.000, B 0.000, C 0.000 }
gfCNCPoint4[14826] = {X 394.3522, Y 59.9221, Z -5.5000, A 0.000, B 0.000, C 0.000 }
gfCNCPoint4[14827] = {X 394.2379, Y 58.9699, Z -5.5000, A 0.000, B 0.000, C 0.000 }
gfCNCPoint4[14828] = {X 394.2377, Y 58.0000, Z -5.5000, A 0.000, B 0.000, C 0.000 }
gfCNCPoint4[14829] = {X 394.3460, Y 57.0387, Z -5.5000, A 0.000, B 0.000, C 0.000 }
gfCNCPoint4[14830] = {X 394.6655, Y 56.1256, Z -5.5000, A 0.000, B 0.000, C 0.000 }
gfCNCPoint4[14831] = {X 395.1802, Y 55.3065, Z -5.5000, A 0.000, B 0.000, C 0.000 }
gfCNCPoint4[14832] = {X 395.8642, Y 54.6225, Z -5.5000, A 0.000, B 0.000, C 0.000 }
gfCNCPoint4[14833] = {X 396.6833, Y 54.1078, Z -5.5000, A 0.000, B 0.000, C 0.000 }
gfCNCPoint4[14834] = {X 397.5964, Y 53.7883, Z -5.5000, A 0.000, B 0.000, C 0.000 }
gfCNCPoint4[14835] = {X 398.5577, Y 53.6800, Z -5.5000, A 0.000, B 0.000, C 0.000 }
gfCNCPoint4[14836] = {X 419.4886, Y 53.6800, Z -5.5000, A 0.000, B 0.000, C 0.000 }
gfCNCPoint4[14837] = {X 420.4499, Y 53.7883, Z -5.5000, A 0.000, B 0.000, C 0.000 }
gfCNCPoint4[14838] = {X 421.3630, Y 54.1078, Z -5.5000, A 0.000, B 0.000, C 0.000 }
gfCNCPoint4[14839] = {X 422.1821, Y 54.6225, Z -5.5000, A 0.000, B 0.000, C 0.000 }
gfCNCPoint4[14840] = {X 422.8661, Y 55.3065, Z -5.5000, A 0.000, B 0.000, C 0.000 }
gfCNCPoint4[14841] = {X 423.3808, Y 56.1256, Z -5.5000, A 0.000, B 0.000, C 0.000 }
gfCNCPoint4[14842] = {X 423.7003, Y 57.0387, Z -5.5000, A 0.000, B 0.000, C 0.000 }
gfCNCPoint4[14843] = {X 423.8086, Y 58.0000, Z -5.5000, A 0.000, B 0.000, C 0.000 }
gfCNCPoint4[14844] = {X 423.8086, Y 58.2319, Z -5.5000, A 0.000, B 0.000, C 0.000 }
gfCNCPoint4[14845] = {X 429.6116, Y 60.4930, Z -5.5000, A 0.000, B 0.000, C 0.000 }
gfCNCPoint4[14846] = {X 457.8584, Y 71.7003, Z -5.5000, A 0.000, B 0.000, C 0.000 }
gfCNCPoint4[14847] = {X 457.8605, Y 63.2123, Z -5.5000, A 0.000, B 0.000, C 0.000 }
gfCNCPoint4[14848] = {X 457.0089, Y 63.0032, Z -5.5000, A 0.000, B 0.000, C 0.000 }
gfCNCPoint4[14849] = {X 456.2170, Y 62.6264, Z -5.5000, A 0.000, B 0.000, C 0.000 }
gfCNCPoint4[14850] = {X 455.5176, Y 62.0974, Z -5.5000, A 0.000, B 0.000, C 0.000 }
gfCNCPoint4[14851] = {X 454.9394, Y 61.4381, Z -5.5000, A 0.000, B 0.000, C 0.000 }
gfCNCPoint4[14852] = {X 454.5062, Y 60.6756, Z -5.5000, A 0.000, B 0.000, C 0.000 }
gfCNCPoint4[14853] = {X 454.2360, Y 59.8414, Z -5.5000, A 0.000, B 0.000, C 0.000 }
gfCNCPoint4[14854] = {X 454.1398, Y 58.9697, Z -5.5000, A 0.000, B 0.000, C 0.000 }
gfCNCPoint4[14855] = {X 454.1396, Y 58.0000, Z -5.5000, A 0.000, B 0.000, C 0.000 }
gfCNCPoint4[14856] = {X 454.2479, Y 57.0387, Z -5.5000, A 0.000, B 0.000, C 0.000 }
gfCNCPoint4[14857] = {X 454.5674, Y 56.1256, Z -5.5000, A 0.000, B 0.000, C 0.000 }
gfCNCPoint4[14858] = {X 455.0821, Y 55.3065, Z -5.5000, A 0.000, B 0.000, C 0.000 }
gfCNCPoint4[14859] = {X 455.7661, Y 54.6225, Z -5.5000, A 0.000, B 0.000, C 0.000 }
gfCNCPoint4[14860] = {X 456.5852, Y 54.1078, Z -5.5000, A 0.000, B 0.000, C 0.000 }
gfCNCPoint4[14861] = {X 457.4983, Y 53.7883, Z -5.5000, A 0.000, B 0.000, C 0.000 }
gfCNCPoint4[14862] = {X 458.4596, Y 53.6800, Z -5.5000, A 0.000, B 0.000, C 0.000 }
gfCNCPoint4[14863] = {X 475.0000, Y 53.6800, Z -5.5000, A 0.000, B 0.000, C 0.000 }
gfCNCPoint4[14864] = {X 475.9613, Y 53.7883, Z -5.5000, A 0.000, B 0.000, C 0.000 }
gfCNCPoint4[14865] = {X 476.8744, Y 54.1078, Z -5.5000, A 0.000, B 0.000, C 0.000 }
gfCNCPoint4[14866] = {X 477.6935, Y 54.6225, Z -5.5000, A 0.000, B 0.000, C 0.000 }
gfCNCPoint4[14867] = {X 478.3775, Y 55.3065, Z -5.5000, A 0.000, B 0.000, C 0.000 }
gfCNCPoint4[14868] = {X 478.8922, Y 56.1256, Z -5.5000, A 0.000, B 0.000, C 0.000 }
gfCNCPoint4[14869] = {X 479.2117, Y 57.0387, Z -5.5000, A 0.000, B 0.000, C 0.000 }
gfCNCPoint4[14870] = {X 479.3200, Y 58.0000, Z -5.5000, A 0.000, B 0.000, C 0.000 }
gfCNCPoint4[14871] = {X 479.3200, Y 58.9342, Z -5.5000, A 0.000, B 0.000, C 0.000 }
gfCNCPoint4[14872] = {X 479.2300, Y 59.8114, Z -5.5000, A 0.000, B 0.000, C 0.000 }
gfCNCPoint4[14873] = {X 478.9637, Y 60.6520, Z -5.5000, A 0.000, B 0.000, C 0.000 }
gfCNCPoint4[14874] = {X 478.5323, Y 61.4211, Z -5.5000, A 0.000, B 0.000, C 0.000 }
gfCNCPoint4[14875] = {X 477.9537, Y 62.0865, Z -5.5000, A 0.000, B 0.000, C 0.000 }
gfCNCPoint4[14876] = {X 477.2521, Y 62.6206, Z -5.5000, A 0.000, B 0.000, C 0.000 }
gfCNCPoint4[14877] = {X 476.4566, Y 63.0011, Z -5.5000, A 0.000, B 0.000, C 0.000 }
gfCNCPoint4[14878] = {X 475.6005, Y 63.2121, Z -5.5000, A 0.000, B 0.000, C 0.000 }
gfCNCPoint4[14879] = {X 475.6009, Y 92.7679, Z -5.5000, A 0.000, B 0.000, C 0.000 }
gfCNCPoint4[14880] = {X 475.9978, Y 92.8671, Z -5.5000, A 0.000, B 0.000, C 0.000 }
gfCNCPoint4[14881] = {X 476.3889, Y 92.9867, Z -5.5000, A 0.000, B 0.000, C 0.000 }
gfCNCPoint4[14882] = {X 477.2003, Y 93.3556, Z -5.5000, A 0.000, B 0.000, C 0.000 }
gfCNCPoint4[14883] = {X 477.9179, Y 93.8841, Z -5.5000, A 0.000, B 0.000, C 0.000 }
gfCNCPoint4[14884] = {X 478.5110, Y 94.5494, Z -5.5000, A 0.000, B 0.000, C 0.000 }
gfCNCPoint4[14885] = {X 478.9539, Y 95.3228, Z -5.5000, A 0.000, B 0.000, C 0.000 }
gfCNCPoint4[14886] = {X 479.2275, Y 96.1711, Z -5.5000, A 0.000, B 0.000, C 0.000 }
gfCNCPoint4[14887] = {X 479.3200, Y 97.0575, Z -5.5000, A 0.000, B 0.000, C 0.000 }
gfCNCPoint4[14888] = {X 479.3200, Y 98.0000, Z -5.5000, A 0.000, B 0.000, C 0.000 }
gfCNCPoint4[14889] = {X 479.2117, Y 98.9613, Z -5.5000, A 0.000, B 0.000, C 0.000 }
gfCNCPoint4[14890] = {X 478.8922, Y 99.8744, Z -5.5000, A 0.000, B 0.000, C 0.000 }
gfCNCPoint4[14891] = {X 478.3775, Y 100.6935, Z -5.5000, A 0.000, B 0.000, C 0.000 }
gfCNCPoint4[14892] = {X 477.6935, Y 101.3775, Z -5.5000, A 0.000, B 0.000, C 0.000 }
gfCNCPoint4[14893] = {X 476.8744, Y 101.8922, Z -5.5000, A 0.000, B 0.000, C 0.000 }
gfCNCPoint4[14894] = {X 475.9613, Y 102.2117, Z -5.5000, A 0.000, B 0.000, C 0.000 }
gfCNCPoint4[14895] = {X 475.0000, Y 102.3200, Z -5.5000, A 0.000, B 0.000, C 0.000 }
gfCNCPoint4[14896] = {X 458.4596, Y 102.3200, Z -5.5000, A 0.000, B 0.000, C 0.000 }
gfCNCPoint4[14897] = {X 457.4983, Y 102.2117, Z -5.5000, A 0.000, B 0.000, C 0.000 }
gfCNCPoint4[14898] = {X 456.5852, Y 101.8922, Z -5.5000, A 0.000, B 0.000, C 0.000 }
gfCNCPoint4[14899] = {X 455.7661, Y 101.3775, Z -5.5000, A 0.000, B 0.000, C 0.000 }
gfCNCPoint4[14900] = {X 455.0821, Y 100.6935, Z -5.5000, A 0.000, B 0.000, C 0.000 }
gfCNCPoint4[14901] = {X 454.5674, Y 99.8744, Z -5.5000, A 0.000, B 0.000, C 0.000 }
gfCNCPoint4[14902] = {X 454.2479, Y 98.9613, Z -5.5000, A 0.000, B 0.000, C 0.000 }
gfCNCPoint4[14903] = {X 454.1396, Y 98.0000, Z -5.5000, A 0.000, B 0.000, C 0.000 }
gfCNCPoint4[14904] = {X 454.1396, Y 97.0659, Z -5.5000, A 0.000, B 0.000, C 0.000 }
gfCNCPoint4[14905] = {X 454.2295, Y 96.1891, Z -5.5000, A 0.000, B 0.000, C 0.000 }
gfCNCPoint4[14906] = {X 454.4955, Y 95.3488, Z -5.5000, A 0.000, B 0.000, C 0.000 }
gfCNCPoint4[14907] = {X 454.9265, Y 94.5800, Z -5.5000, A 0.000, B 0.000, C 0.000 }
gfCNCPoint4[14908] = {X 455.5046, Y 93.9147, Z -5.5000, A 0.000, B 0.000, C 0.000 }
gfCNCPoint4[14909] = {X 456.2057, Y 93.3805, Z -5.5000, A 0.000, B 0.000, C 0.000 }
gfCNCPoint4[14910] = {X 457.0006, Y 92.9998, Z -5.5000, A 0.000, B 0.000, C 0.000 }
gfCNCPoint4[14911] = {X 457.8563, Y 92.7883, Z -5.5000, A 0.000, B 0.000, C 0.000 }
gfCNCPoint4[14912] = {X 457.8563, Y 85.5950, Z -5.5000, A 0.000, B 0.000, C 0.000 }
gfCNCPoint4[14913] = {X 444.8595, Y 80.5002, Z -5.5000, A 0.000, B 0.000, C 0.000 }
gfCNCPoint4[14914] = {X 420.0237, Y 96.5883, Z -5.5000, A 0.000, B 0.000, C 0.000 }
gfCNCPoint4[14915] = {X 420.0267, Y 97.0649, Z -5.5000, A 0.000, B 0.000, C 0.000 }
gfCNCPoint4[14916] = {X 420.0267, Y 98.0000, Z -5.5000, A 0.000, B 0.000, C 0.000 }
gfCNCPoint4[14917] = {X 419.9184, Y 98.9613, Z -5.5000, A 0.000, B 0.000, C 0.000 }
gfCNCPoint4[14918] = {X 419.5989, Y 99.8744, Z -5.5000, A 0.000, B 0.000, C 0.000 }
gfCNCPoint4[14919] = {X 419.0842, Y 100.6935, Z -5.5000, A 0.000, B 0.000, C 0.000 }
gfCNCPoint4[14920] = {X 418.4002, Y 101.3775, Z -5.5000, A 0.000, B 0.000, C 0.000 }
gfCNCPoint4[14921] = {X 417.5811, Y 101.8922, Z -5.5000, A 0.000, B 0.000, C 0.000 }
gfCNCPoint4[14922] = {X 416.6680, Y 102.2117, Z -5.5000, A 0.000, B 0.000, C 0.000 }
gfCNCPoint4[14923] = {X 415.7067, Y 102.3200, Z -5.5000, A 0.000, B 0.000, C 0.000 }
gfCNCPoint4[14924] = {X 396.4059, Y 102.3200, Z -5.5000, A 0.000, B 0.000, C 0.000 }
gfCNCPoint4[14925] = {X 395.4447, Y 102.2117, Z -5.5000, A 0.000, B 0.000, C 0.000 }
gfCNCPoint4[14926] = {X 394.5316, Y 101.8922, Z -5.5000, A 0.000, B 0.000, C 0.000 }
gfCNCPoint4[14927] = {X 393.7125, Y 101.3775, Z -5.5000, A 0.000, B 0.000, C 0.000 }
gfCNCPoint4[14928] = {X 393.0284, Y 100.6935, Z -5.5000, A 0.000, B 0.000, C 0.000 }
gfCNCPoint4[14929] = {X 392.5138, Y 99.8744, Z -5.5000, A 0.000, B 0.000, C 0.000 }
gfCNCPoint4[14930] = {X 392.1943, Y 98.9613, Z -5.5000, A 0.000, B 0.000, C 0.000 }
gfCNCPoint4[14931] = {X 392.0859, Y 98.0000, Z -5.5000, A 0.000, B 0.000, C 0.000 }
gfCNCPoint4[14932] = {X 392.0859, Y 97.0659, Z -5.5000, A 0.000, B 0.000, C 0.000 }
gfCNCPoint4[14933] = {X 392.1947, Y 96.1026, Z -5.5000, A 0.000, B 0.000, C 0.000 }
gfCNCPoint4[14934] = {X 392.5156, Y 95.1877, Z -5.5000, A 0.000, B 0.000, C 0.000 }
gfCNCPoint4[14935] = {X 393.0324, Y 94.3675, Z -5.5000, A 0.000, B 0.000, C 0.000 }
gfCNCPoint4[14936] = {X 393.7191, Y 93.6831, Z -5.5000, A 0.000, B 0.000, C 0.000 }
gfCNCPoint4[14937] = {X 394.5412, Y 93.1691, Z -5.5000, A 0.000, B 0.000, C 0.000 }
gfCNCPoint4[14938] = {X 395.4571, Y 92.8514, Z -5.5000, A 0.000, B 0.000, C 0.000 }
gfCNCPoint4[14939] = {X 396.4208, Y 92.7460, Z -5.5000, A 0.000, B 0.000, C 0.000 }
gfCNCPoint4[14940] = {X 397.3588, Y 92.7029, Z -5.5000, A 0.000, B 0.000, C 0.000 }
gfCNCPoint4[14941] = {X 398.2935, Y 92.6140, Z -5.5000, A 0.000, B 0.000, C 0.000 }
gfCNCPoint4[14942] = {X 398.9444, Y 92.4560, Z -5.5000, A 0.000, B 0.000, C 0.000 }
gfCNCPoint4[14943] = {X 399.5438, Y 92.1572, Z -5.5000, A 0.000, B 0.000, C 0.000 }
gfCNCPoint4[14944] = {X 413.7990, Y 83.0284, Z -5.5000, A 0.000, B 0.000, C 0.000 }
gfCNCPoint4[14945] = {X 411.6418, Y 79.6599, Z -5.5000, A 0.000, B 0.000, C 0.000 }
gfCNCPoint4[14946] = {X 413.8421, Y 83.0958, Z -5.5000, A 0.000, B 0.000, C 0.000 }
gfCNCPoint4[14947] = {X 428.2294, Y 73.8824, Z -5.5000, A 0.000, B 0.000, C 0.000 }
gfCNCPoint4[14948] = {X 403.7848, Y 64.2917, Z -5.5000, A 0.000, B 0.000, C 0.000 }
gfCNCPoint4[14949] = {X 402.0800, Y 63.7274, Z -5.5000, A 0.000, B 0.000, C 0.000 }
gfCNCPoint4[14950] = {X 400.3236, Y 63.3533, Z -5.5000, A 0.000, B 0.000, C 0.000 }
gfCNCPoint4[14951] = {X 398.5368, Y 63.1740, Z -5.5000, A 0.000, B 0.000, C 0.000 }
gfCNCPoint4[14952] = {X 397.6017, Y 63.0649, Z -5.5000, A 0.000, B 0.000, C 0.000 }
gfCNCPoint4[14953] = {X 396.7137, Y 62.7521, Z -5.5000, A 0.000, B 0.000, C 0.000 }
gfCNCPoint4[14954] = {X 395.9166, Y 62.2510, Z -5.5000, A 0.000, B 0.000, C 0.000 }
gfCNCPoint4[14955] = {X 395.2497, Y 61.5864, Z -5.5000, A 0.000, B 0.000, C 0.000 }
gfCNCPoint4[14956] = {X 394.7460, Y 60.7910, Z -5.5000, A 0.000, B 0.000, C 0.000 }
gfCNCPoint4[14957] = {X 394.4302, Y 59.9040, Z -5.5000, A 0.000, B 0.000, C 0.000 }
gfCNCPoint4[14958] = {X 394.3179, Y 58.9693, Z -5.5000, A 0.000, B 0.000, C 0.000 }
gfCNCPoint4[14959] = {X 394.3177, Y 58.0000, Z -5.5000, A 0.000, B 0.000, C 0.000 }
gfCNCPoint4[14960] = {X 394.4240, Y 57.0565, Z -5.5000, A 0.000, B 0.000, C 0.000 }
gfCNCPoint4[14961] = {X 394.7376, Y 56.1603, Z -5.5000, A 0.000, B 0.000, C 0.000 }
gfCNCPoint4[14962] = {X 395.2428, Y 55.3564, Z -5.5000, A 0.000, B 0.000, C 0.000 }
gfCNCPoint4[14963] = {X 395.9141, Y 54.6850, Z -5.5000, A 0.000, B 0.000, C 0.000 }
gfCNCPoint4[14964] = {X 396.7181, Y 54.1799, Z -5.5000, A 0.000, B 0.000, C 0.000 }
gfCNCPoint4[14965] = {X 397.6142, Y 53.8663, Z -5.5000, A 0.000, B 0.000, C 0.000 }
gfCNCPoint4[14966] = {X 398.5577, Y 53.7600, Z -5.5000, A 0.000, B 0.000, C 0.000 }
gfCNCPoint4[14967] = {X 419.4886, Y 53.7600, Z -5.5000, A 0.000, B 0.000, C 0.000 }
gfCNCPoint4[14968] = {X 420.4321, Y 53.8663, Z -5.5000, A 0.000, B 0.000, C 0.000 }
gfCNCPoint4[14969] = {X 421.3283, Y 54.1799, Z -5.5000, A 0.000, B 0.000, C 0.000 }
gfCNCPoint4[14970] = {X 422.1322, Y 54.6850, Z -5.5000, A 0.000, B 0.000, C 0.000 }
gfCNCPoint4[14971] = {X 422.8036, Y 55.3564, Z -5.5000, A 0.000, B 0.000, C 0.000 }
gfCNCPoint4[14972] = {X 423.3087, Y 56.1603, Z -5.5000, A 0.000, B 0.000, C 0.000 }
gfCNCPoint4[14973] = {X 423.6223, Y 57.0565, Z -5.5000, A 0.000, B 0.000, C 0.000 }
gfCNCPoint4[14974] = {X 423.7286, Y 58.0000, Z -5.5000, A 0.000, B 0.000, C 0.000 }
gfCNCPoint4[14975] = {X 423.7286, Y 58.2866, Z -5.5000, A 0.000, B 0.000, C 0.000 }
gfCNCPoint4[14976] = {X 429.5823, Y 60.5675, Z -5.5000, A 0.000, B 0.000, C 0.000 }
gfCNCPoint4[14977] = {X 457.9384, Y 71.8181, Z -5.5000, A 0.000, B 0.000, C 0.000 }
gfCNCPoint4[14978] = {X 457.9406, Y 63.1422, Z -5.5000, A 0.000, B 0.000, C 0.000 }
gfCNCPoint4[14979] = {X 457.0920, Y 62.9475, Z -5.5000, A 0.000, B 0.000, C 0.000 }
gfCNCPoint4[14980] = {X 456.3012, Y 62.5835, Z -5.5000, A 0.000, B 0.000, C 0.000 }
gfCNCPoint4[14981] = {X 455.6013, Y 62.0658, Z -5.5000, A 0.000, B 0.000, C 0.000 }
gfCNCPoint4[14982] = {X 455.0219, Y 61.4160, Z -5.5000, A 0.000, B 0.000, C 0.000 }
gfCNCPoint4[14983] = {X 454.5875, Y 60.6616, Z -5.5000, A 0.000, B 0.000, C 0.000 }
gfCNCPoint4[14984] = {X 454.3163, Y 59.8343, Z -5.5000, A 0.000, B 0.000, C 0.000 }
gfCNCPoint4[14985] = {X 454.2197, Y 58.9691, Z -5.5000, A 0.000, B 0.000, C 0.000 }
gfCNCPoint4[14986] = {X 454.2196, Y 58.0000, Z -5.5000, A 0.000, B 0.000, C 0.000 }
gfCNCPoint4[14987] = {X 454.3259, Y 57.0565, Z -5.5000, A 0.000, B 0.000, C 0.000 }
gfCNCPoint4[14988] = {X 454.6395, Y 56.1603, Z -5.5000, A 0.000, B 0.000, C 0.000 }
gfCNCPoint4[14989] = {X 455.1446, Y 55.3564, Z -5.5000, A 0.000, B 0.000, C 0.000 }
gfCNCPoint4[14990] = {X 455.8160, Y 54.6850, Z -5.5000, A 0.000, B 0.000, C 0.000 }
gfCNCPoint4[14991] = {X 456.6199, Y 54.1799, Z -5.5000, A 0.000, B 0.000, C 0.000 }
gfCNCPoint4[14992] = {X 457.5161, Y 53.8663, Z -5.5000, A 0.000, B 0.000, C 0.000 }
gfCNCPoint4[14993] = {X 458.4596, Y 53.7600, Z -5.5000, A 0.000, B 0.000, C 0.000 }
gfCNCPoint4[14994] = {X 475.0000, Y 53.7600, Z -5.5000, A 0.000, B 0.000, C 0.000 }
gfCNCPoint4[14995] = {X 475.9435, Y 53.8663, Z -5.5000, A 0.000, B 0.000, C 0.000 }
gfCNCPoint4[14996] = {X 476.8397, Y 54.1799, Z -5.5000, A 0.000, B 0.000, C 0.000 }
gfCNCPoint4[14997] = {X 477.6436, Y 54.6850, Z -5.5000, A 0.000, B 0.000, C 0.000 }
gfCNCPoint4[14998] = {X 478.3150, Y 55.3564, Z -5.5000, A 0.000, B 0.000, C 0.000 }
gfCNCPoint4[14999] = {X 478.8201, Y 56.1603, Z -5.5000, A 0.000, B 0.000, C 0.000 }
gfCNCPoint4[15000] = {X 479.1337, Y 57.0565, Z -5.5000, A 0.000, B 0.000, C 0.000 }
gfCNCPoint4[15001] = {X 479.2400, Y 58.0000, Z -5.5000, A 0.000, B 0.000, C 0.000 }
gfCNCPoint4[15002] = {X 479.2400, Y 58.9342, Z -5.5000, A 0.000, B 0.000, C 0.000 }
gfCNCPoint4[15003] = {X 479.1496, Y 59.8049, Z -5.5000, A 0.000, B 0.000, C 0.000 }
gfCNCPoint4[15004] = {X 478.8824, Y 60.6384, Z -5.5000, A 0.000, B 0.000, C 0.000 }
gfCNCPoint4[15005] = {X 478.4497, Y 61.3993, Z -5.5000, A 0.000, B 0.000, C 0.000 }
gfCNCPoint4[15006] = {X 477.8699, Y 62.0551, Z -5.5000, A 0.000, B 0.000, C 0.000 }
gfCNCPoint4[15007] = {X 477.1679, Y 62.5779, Z -5.5000, A 0.000, B 0.000, C 0.000 }
gfCNCPoint4[15008] = {X 476.3735, Y 62.9455, Z -5.5000, A 0.000, B 0.000, C 0.000 }
gfCNCPoint4[15009] = {X 475.5205, Y 63.1420, Z -5.5000, A 0.000, B 0.000, C 0.000 }
gfCNCPoint4[15010] = {X 475.5209, Y 92.8323, Z -5.5000, A 0.000, B 0.000, C 0.000 }
gfCNCPoint4[15011] = {X 475.9455, Y 92.9356, Z -5.5000, A 0.000, B 0.000, C 0.000 }
gfCNCPoint4[15012] = {X 476.3635, Y 93.0626, Z -5.5000, A 0.000, B 0.000, C 0.000 }
gfCNCPoint4[15013] = {X 477.1598, Y 93.4246, Z -5.5000, A 0.000, B 0.000, C 0.000 }
gfCNCPoint4[15014] = {X 477.8641, Y 93.9432, Z -5.5000, A 0.000, B 0.000, C 0.000 }
gfCNCPoint4[15015] = {X 478.4461, Y 94.5961, Z -5.5000, A 0.000, B 0.000, C 0.000 }
gfCNCPoint4[15016] = {X 478.8807, Y 95.3552, Z -5.5000, A 0.000, B 0.000, C 0.000 }
gfCNCPoint4[15017] = {X 479.1492, Y 96.1876, Z -5.5000, A 0.000, B 0.000, C 0.000 }
gfCNCPoint4[15018] = {X 479.2400, Y 97.0575, Z -5.5000, A 0.000, B 0.000, C 0.000 }
gfCNCPoint4[15019] = {X 479.2400, Y 98.0000, Z -5.5000, A 0.000, B 0.000, C 0.000 }
gfCNCPoint4[15020] = {X 479.1337, Y 98.9435, Z -5.5000, A 0.000, B 0.000, C 0.000 }
gfCNCPoint4[15021] = {X 478.8201, Y 99.8397, Z -5.5000, A 0.000, B 0.000, C 0.000 }
gfCNCPoint4[15022] = {X 478.3150, Y 100.6436, Z -5.5000, A 0.000, B 0.000, C 0.000 }
gfCNCPoint4[15023] = {X 477.6436, Y 101.3150, Z -5.5000, A 0.000, B 0.000, C 0.000 }
gfCNCPoint4[15024] = {X 476.8397, Y 101.8201, Z -5.5000, A 0.000, B 0.000, C 0.000 }
gfCNCPoint4[15025] = {X 475.9435, Y 102.1337, Z -5.5000, A 0.000, B 0.000, C 0.000 }
gfCNCPoint4[15026] = {X 475.0000, Y 102.2400, Z -5.5000, A 0.000, B 0.000, C 0.000 }
gfCNCPoint4[15027] = {X 458.4596, Y 102.2400, Z -5.5000, A 0.000, B 0.000, C 0.000 }
gfCNCPoint4[15028] = {X 457.5161, Y 102.1337, Z -5.5000, A 0.000, B 0.000, C 0.000 }
gfCNCPoint4[15029] = {X 456.6199, Y 101.8201, Z -5.5000, A 0.000, B 0.000, C 0.000 }
gfCNCPoint4[15030] = {X 455.8160, Y 101.3150, Z -5.5000, A 0.000, B 0.000, C 0.000 }
gfCNCPoint4[15031] = {X 455.1446, Y 100.6436, Z -5.5000, A 0.000, B 0.000, C 0.000 }
gfCNCPoint4[15032] = {X 454.6395, Y 99.8397, Z -5.5000, A 0.000, B 0.000, C 0.000 }
gfCNCPoint4[15033] = {X 454.3259, Y 98.9435, Z -5.5000, A 0.000, B 0.000, C 0.000 }
gfCNCPoint4[15034] = {X 454.2196, Y 98.0000, Z -5.5000, A 0.000, B 0.000, C 0.000 }
gfCNCPoint4[15035] = {X 454.2196, Y 97.0659, Z -5.5000, A 0.000, B 0.000, C 0.000 }
gfCNCPoint4[15036] = {X 454.3099, Y 96.1957, Z -5.5000, A 0.000, B 0.000, C 0.000 }
gfCNCPoint4[15037] = {X 454.5769, Y 95.3624, Z -5.5000, A 0.000, B 0.000, C 0.000 }
gfCNCPoint4[15038] = {X 455.0092, Y 94.6018, Z -5.5000, A 0.000, B 0.000, C 0.000 }
gfCNCPoint4[15039] = {X 455.5884, Y 93.9460, Z -5.5000, A 0.000, B 0.000, C 0.000 }
gfCNCPoint4[15040] = {X 456.2899, Y 93.4231, Z -5.5000, A 0.000, B 0.000, C 0.000 }
gfCNCPoint4[15041] = {X 457.0838, Y 93.0553, Z -5.5000, A 0.000, B 0.000, C 0.000 }
gfCNCPoint4[15042] = {X 457.9363, Y 92.8584, Z -5.5000, A 0.000, B 0.000, C 0.000 }
gfCNCPoint4[15043] = {X 457.9363, Y 85.5404, Z -5.5000, A 0.000, B 0.000, C 0.000 }
gfCNCPoint4[15044] = {X 444.8504, Y 80.4107, Z -5.5000, A 0.000, B 0.000, C 0.000 }
gfCNCPoint4[15045] = {X 419.9434, Y 96.5450, Z -5.5000, A 0.000, B 0.000, C 0.000 }
gfCNCPoint4[15046] = {X 419.9467, Y 97.0651, Z -5.5000, A 0.000, B 0.000, C 0.000 }
gfCNCPoint4[15047] = {X 419.9467, Y 98.0000, Z -5.5000, A 0.000, B 0.000, C 0.000 }
gfCNCPoint4[15048] = {X 419.8404, Y 98.9435, Z -5.5000, A 0.000, B 0.000, C 0.000 }
gfCNCPoint4[15049] = {X 419.5268, Y 99.8397, Z -5.5000, A 0.000, B 0.000, C 0.000 }
gfCNCPoint4[15050] = {X 419.0217, Y 100.6436, Z -5.5000, A 0.000, B 0.000, C 0.000 }
gfCNCPoint4[15051] = {X 418.3503, Y 101.3150, Z -5.5000, A 0.000, B 0.000, C 0.000 }
gfCNCPoint4[15052] = {X 417.5464, Y 101.8201, Z -5.5000, A 0.000, B 0.000, C 0.000 }
gfCNCPoint4[15053] = {X 416.6502, Y 102.1337, Z -5.5000, A 0.000, B 0.000, C 0.000 }
gfCNCPoint4[15054] = {X 415.7067, Y 102.2400, Z -5.5000, A 0.000, B 0.000, C 0.000 }
gfCNCPoint4[15055] = {X 396.4059, Y 102.2400, Z -5.5000, A 0.000, B 0.000, C 0.000 }
gfCNCPoint4[15056] = {X 395.4625, Y 102.1337, Z -5.5000, A 0.000, B 0.000, C 0.000 }
gfCNCPoint4[15057] = {X 394.5663, Y 101.8201, Z -5.5000, A 0.000, B 0.000, C 0.000 }
gfCNCPoint4[15058] = {X 393.7624, Y 101.3150, Z -5.5000, A 0.000, B 0.000, C 0.000 }
gfCNCPoint4[15059] = {X 393.0910, Y 100.6436, Z -5.5000, A 0.000, B 0.000, C 0.000 }
gfCNCPoint4[15060] = {X 392.5858, Y 99.8397, Z -5.5000, A 0.000, B 0.000, C 0.000 }
gfCNCPoint4[15061] = {X 392.2723, Y 98.9435, Z -5.5000, A 0.000, B 0.000, C 0.000 }
gfCNCPoint4[15062] = {X 392.1659, Y 98.0000, Z -5.5000, A 0.000, B 0.000, C 0.000 }
gfCNCPoint4[15063] = {X 392.1659, Y 97.0659, Z -5.5000, A 0.000, B 0.000, C 0.000 }
gfCNCPoint4[15064] = {X 392.2728, Y 96.1203, Z -5.5000, A 0.000, B 0.000, C 0.000 }
gfCNCPoint4[15065] = {X 392.5878, Y 95.2222, Z -5.5000, A 0.000, B 0.000, C 0.000 }
gfCNCPoint4[15066] = {X 393.0952, Y 94.4171, Z -5.5000, A 0.000, B 0.000, C 0.000 }
gfCNCPoint4[15067] = {X 393.7693, Y 93.7454, Z -5.5000, A 0.000, B 0.000, C 0.000 }
gfCNCPoint4[15068] = {X 394.5763, Y 93.2410, Z -5.5000, A 0.000, B 0.000, C 0.000 }
gfCNCPoint4[15069] = {X 395.4755, Y 92.9293, Z -5.5000, A 0.000, B 0.000, C 0.000 }
gfCNCPoint4[15070] = {X 396.4216, Y 92.8260, Z -5.5000, A 0.000, B 0.000, C 0.000 }
gfCNCPoint4[15071] = {X 397.3641, Y 92.7827, Z -5.5000, A 0.000, B 0.000, C 0.000 }
gfCNCPoint4[15072] = {X 398.3033, Y 92.6934, Z -5.5000, A 0.000, B 0.000, C 0.000 }
gfCNCPoint4[15073] = {X 398.9717, Y 92.5312, Z -5.5000, A 0.000, B 0.000, C 0.000 }
gfCNCPoint4[15074] = {X 399.5872, Y 92.2244, Z -5.5000, A 0.000, B 0.000, C 0.000 }
gfCNCPoint4[15075] = {X 413.8421, Y 83.0958, Z -5.5000, A 0.000, B 0.000, C 0.000 }
gfCNCPoint4[15076] = {X 411.6850, Y 79.7273, Z -5.5000, A 0.000, B 0.000, C 0.000 }
gfCNCPoint4[15077] = {X 413.8852, Y 83.1631, Z -5.5000, A 0.000, B 0.000, C 0.000 }
gfCNCPoint4[15078] = {X 428.4046, Y 73.8652, Z -5.5000, A 0.000, B 0.000, C 0.000 }
gfCNCPoint4[15079] = {X 403.8141, Y 64.2173, Z -5.5000, A 0.000, B 0.000, C 0.000 }
gfCNCPoint4[15080] = {X 402.1004, Y 63.6500, Z -5.5000, A 0.000, B 0.000, C 0.000 }
gfCNCPoint4[15081] = {X 400.3349, Y 63.2741, Z -5.5000, A 0.000, B 0.000, C 0.000 }
gfCNCPoint4[15082] = {X 398.5388, Y 63.0940, Z -5.5000, A 0.000, B 0.000, C 0.000 }
gfCNCPoint4[15083] = {X 397.6210, Y 62.9872, Z -5.5000, A 0.000, B 0.000, C 0.000 }
gfCNCPoint4[15084] = {X 396.7495, Y 62.6805, Z -5.5000, A 0.000, B 0.000, C 0.000 }
gfCNCPoint4[15085] = {X 395.9671, Y 62.1890, Z -5.5000, A 0.000, B 0.000, C 0.000 }
gfCNCPoint4[15086] = {X 395.3126, Y 61.5369, Z -5.5000, A 0.000, B 0.000, C 0.000 }
gfCNCPoint4[15087] = {X 394.8181, Y 60.7564, Z -5.5000, A 0.000, B 0.000, C 0.000 }
gfCNCPoint4[15088] = {X 394.5081, Y 59.8860, Z -5.5000, A 0.000, B 0.000, C 0.000 }
gfCNCPoint4[15089] = {X 394.3979, Y 58.9686, Z -5.5000, A 0.000, B 0.000, C 0.000 }
gfCNCPoint4[15090] = {X 394.3977, Y 58.0000, Z -5.5000, A 0.000, B 0.000, C 0.000 }
gfCNCPoint4[15091] = {X 394.5020, Y 57.0743, Z -5.5000, A 0.000, B 0.000, C 0.000 }
gfCNCPoint4[15092] = {X 394.8097, Y 56.1950, Z -5.5000, A 0.000, B 0.000, C 0.000 }
gfCNCPoint4[15093] = {X 395.3053, Y 55.4063, Z -5.5000, A 0.000, B 0.000, C 0.000 }
gfCNCPoint4[15094] = {X 395.9640, Y 54.7476, Z -5.5000, A 0.000, B 0.000, C 0.000 }
gfCNCPoint4[15095] = {X 396.7528, Y 54.2520, Z -5.5000, A 0.000, B 0.000, C 0.000 }
gfCNCPoint4[15096] = {X 397.6320, Y 53.9443, Z -5.5000, A 0.000, B 0.000, C 0.000 }
gfCNCPoint4[15097] = {X 398.5577, Y 53.8400, Z -5.5000, A 0.000, B 0.000, C 0.000 }
gfCNCPoint4[15098] = {X 419.4886, Y 53.8400, Z -5.5000, A 0.000, B 0.000, C 0.000 }
gfCNCPoint4[15099] = {X 420.4143, Y 53.9443, Z -5.5000, A 0.000, B 0.000, C 0.000 }
gfCNCPoint4[15100] = {X 421.2936, Y 54.2520, Z -5.5000, A 0.000, B 0.000, C 0.000 }
gfCNCPoint4[15101] = {X 422.0823, Y 54.7476, Z -5.5000, A 0.000, B 0.000, C 0.000 }
gfCNCPoint4[15102] = {X 422.7410, Y 55.4063, Z -5.5000, A 0.000, B 0.000, C 0.000 }
gfCNCPoint4[15103] = {X 423.2366, Y 56.1950, Z -5.5000, A 0.000, B 0.000, C 0.000 }
gfCNCPoint4[15104] = {X 423.5443, Y 57.0743, Z -5.5000, A 0.000, B 0.000, C 0.000 }
gfCNCPoint4[15105] = {X 423.6486, Y 58.0000, Z -5.5000, A 0.000, B 0.000, C 0.000 }
gfCNCPoint4[15106] = {X 423.6486, Y 58.3413, Z -5.5000, A 0.000, B 0.000, C 0.000 }
gfCNCPoint4[15107] = {X 429.5531, Y 60.6419, Z -5.5000, A 0.000, B 0.000, C 0.000 }
gfCNCPoint4[15108] = {X 458.0184, Y 71.9359, Z -5.5000, A 0.000, B 0.000, C 0.000 }
gfCNCPoint4[15109] = {X 458.0206, Y 63.0708, Z -5.5000, A 0.000, B 0.000, C 0.000 }
gfCNCPoint4[15110] = {X 457.9181, Y 63.0587, Z -5.5000, A 0.000, B 0.000, C 0.000 }
gfCNCPoint4[15111] = {X 457.8159, Y 63.0440, Z -5.5000, A 0.000, B 0.000, C 0.000 }
gfCNCPoint4[15112] = {X 456.8785, Y 62.7819, Z -5.5000, A 0.000, B 0.000, C 0.000 }
gfCNCPoint4[15113] = {X 456.0276, Y 62.3091, Z -5.5000, A 0.000, B 0.000, C 0.000 }
gfCNCPoint4[15114] = {X 455.3098, Y 61.6515, Z -5.5000, A 0.000, B 0.000, C 0.000 }
gfCNCPoint4[15115] = {X 454.7646, Y 60.8452, Z -5.5000, A 0.000, B 0.000, C 0.000 }
gfCNCPoint4[15116] = {X 454.4216, Y 59.9342, Z -5.5000, A 0.000, B 0.000, C 0.000 }
gfCNCPoint4[15117] = {X 454.2997, Y 58.9684, Z -5.5000, A 0.000, B 0.000, C 0.000 }
gfCNCPoint4[15118] = {X 454.2996, Y 58.0000, Z -5.5000, A 0.000, B 0.000, C 0.000 }
gfCNCPoint4[15119] = {X 454.4039, Y 57.0743, Z -5.5000, A 0.000, B 0.000, C 0.000 }
gfCNCPoint4[15120] = {X 454.7116, Y 56.1950, Z -5.5000, A 0.000, B 0.000, C 0.000 }
gfCNCPoint4[15121] = {X 455.2072, Y 55.4063, Z -5.5000, A 0.000, B 0.000, C 0.000 }
gfCNCPoint4[15122] = {X 455.8659, Y 54.7476, Z -5.5000, A 0.000, B 0.000, C 0.000 }
gfCNCPoint4[15123] = {X 456.6546, Y 54.2520, Z -5.5000, A 0.000, B 0.000, C 0.000 }
gfCNCPoint4[15124] = {X 457.5339, Y 53.9443, Z -5.5000, A 0.000, B 0.000, C 0.000 }
gfCNCPoint4[15125] = {X 458.4596, Y 53.8400, Z -5.5000, A 0.000, B 0.000, C 0.000 }
gfCNCPoint4[15126] = {X 475.0000, Y 53.8400, Z -5.5000, A 0.000, B 0.000, C 0.000 }
gfCNCPoint4[15127] = {X 475.9257, Y 53.9443, Z -5.5000, A 0.000, B 0.000, C 0.000 }
gfCNCPoint4[15128] = {X 476.8050, Y 54.2520, Z -5.5000, A 0.000, B 0.000, C 0.000 }
gfCNCPoint4[15129] = {X 477.5937, Y 54.7476, Z -5.5000, A 0.000, B 0.000, C 0.000 }
gfCNCPoint4[15130] = {X 478.2524, Y 55.4063, Z -5.5000, A 0.000, B 0.000, C 0.000 }
gfCNCPoint4[15131] = {X 478.7480, Y 56.1950, Z -5.5000, A 0.000, B 0.000, C 0.000 }
gfCNCPoint4[15132] = {X 479.0557, Y 57.0743, Z -5.5000, A 0.000, B 0.000, C 0.000 }
gfCNCPoint4[15133] = {X 479.1600, Y 58.0000, Z -5.5000, A 0.000, B 0.000, C 0.000 }
gfCNCPoint4[15134] = {X 479.1600, Y 58.9342, Z -5.5000, A 0.000, B 0.000, C 0.000 }
gfCNCPoint4[15135] = {X 479.0692, Y 59.7983, Z -5.5000, A 0.000, B 0.000, C 0.000 }
gfCNCPoint4[15136] = {X 478.8010, Y 60.6247, Z -5.5000, A 0.000, B 0.000, C 0.000 }
gfCNCPoint4[15137] = {X 478.3669, Y 61.3774, Z -5.5000, A 0.000, B 0.000, C 0.000 }
gfCNCPoint4[15138] = {X 477.7859, Y 62.0234, Z -5.5000, A 0.000, B 0.000, C 0.000 }
gfCNCPoint4[15139] = {X 477.0835, Y 62.5347, Z -5.5000, A 0.000, B 0.000, C 0.000 }
gfCNCPoint4[15140] = {X 476.2901, Y 62.8890, Z -5.5000, A 0.000, B 0.000, C 0.000 }
gfCNCPoint4[15141] = {X 475.4405, Y 63.0707, Z -5.5000, A 0.000, B 0.000, C 0.000 }
gfCNCPoint4[15142] = {X 475.4409, Y 92.8973, Z -5.5000, A 0.000, B 0.000, C 0.000 }
gfCNCPoint4[15143] = {X 475.8932, Y 93.0044, Z -5.5000, A 0.000, B 0.000, C 0.000 }
gfCNCPoint4[15144] = {X 476.3382, Y 93.1384, Z -5.5000, A 0.000, B 0.000, C 0.000 }
gfCNCPoint4[15145] = {X 477.1193, Y 93.4936, Z -5.5000, A 0.000, B 0.000, C 0.000 }
gfCNCPoint4[15146] = {X 477.8102, Y 94.0024, Z -5.5000, A 0.000, B 0.000, C 0.000 }
gfCNCPoint4[15147] = {X 478.3811, Y 94.6429, Z -5.5000, A 0.000, B 0.000, C 0.000 }
gfCNCPoint4[15148] = {X 478.8075, Y 95.3875, Z -5.5000, A 0.000, B 0.000, C 0.000 }
gfCNCPoint4[15149] = {X 479.0709, Y 96.2041, Z -5.5000, A 0.000, B 0.000, C 0.000 }
gfCNCPoint4[15150] = {X 479.1600, Y 97.0575, Z -5.5000, A 0.000, B 0.000, C 0.000 }
gfCNCPoint4[15151] = {X 479.1600, Y 98.0000, Z -5.5000, A 0.000, B 0.000, C 0.000 }
gfCNCPoint4[15152] = {X 479.0557, Y 98.9257, Z -5.5000, A 0.000, B 0.000, C 0.000 }
gfCNCPoint4[15153] = {X 478.7480, Y 99.8050, Z -5.5000, A 0.000, B 0.000, C 0.000 }
gfCNCPoint4[15154] = {X 478.2524, Y 100.5937, Z -5.5000, A 0.000, B 0.000, C 0.000 }
gfCNCPoint4[15155] = {X 477.5937, Y 101.2524, Z -5.5000, A 0.000, B 0.000, C 0.000 }
gfCNCPoint4[15156] = {X 476.8050, Y 101.7480, Z -5.5000, A 0.000, B 0.000, C 0.000 }
gfCNCPoint4[15157] = {X 475.9257, Y 102.0557, Z -5.5000, A 0.000, B 0.000, C 0.000 }
gfCNCPoint4[15158] = {X 475.0000, Y 102.1600, Z -5.5000, A 0.000, B 0.000, C 0.000 }
gfCNCPoint4[15159] = {X 458.4596, Y 102.1600, Z -5.5000, A 0.000, B 0.000, C 0.000 }
gfCNCPoint4[15160] = {X 457.5339, Y 102.0557, Z -5.5000, A 0.000, B 0.000, C 0.000 }
gfCNCPoint4[15161] = {X 456.6546, Y 101.7480, Z -5.5000, A 0.000, B 0.000, C 0.000 }
gfCNCPoint4[15162] = {X 455.8659, Y 101.2524, Z -5.5000, A 0.000, B 0.000, C 0.000 }
gfCNCPoint4[15163] = {X 455.2072, Y 100.5937, Z -5.5000, A 0.000, B 0.000, C 0.000 }
gfCNCPoint4[15164] = {X 454.7116, Y 99.8050, Z -5.5000, A 0.000, B 0.000, C 0.000 }
gfCNCPoint4[15165] = {X 454.4039, Y 98.9257, Z -5.5000, A 0.000, B 0.000, C 0.000 }
gfCNCPoint4[15166] = {X 454.2996, Y 98.0000, Z -5.5000, A 0.000, B 0.000, C 0.000 }
gfCNCPoint4[15167] = {X 454.2996, Y 97.0659, Z -5.5000, A 0.000, B 0.000, C 0.000 }
gfCNCPoint4[15168] = {X 454.3903, Y 96.2022, Z -5.5000, A 0.000, B 0.000, C 0.000 }
gfCNCPoint4[15169] = {X 454.6583, Y 95.3761, Z -5.5000, A 0.000, B 0.000, C 0.000 }
gfCNCPoint4[15170] = {X 455.0920, Y 94.6237, Z -5.5000, A 0.000, B 0.000, C 0.000 }
gfCNCPoint4[15171] = {X 455.6724, Y 93.9777, Z -5.5000, A 0.000, B 0.000, C 0.000 }
gfCNCPoint4[15172] = {X 456.3743, Y 93.4663, Z -5.5000, A 0.000, B 0.000, C 0.000 }
gfCNCPoint4[15173] = {X 457.1672, Y 93.1118, Z -5.5000, A 0.000, B 0.000, C 0.000 }
gfCNCPoint4[15174] = {X 458.0163, Y 92.9296, Z -5.5000, A 0.000, B 0.000, C 0.000 }
gfCNCPoint4[15175] = {X 458.0163, Y 85.4858, Z -5.5000, A 0.000, B 0.000, C 0.000 }
gfCNCPoint4[15176] = {X 444.8414, Y 80.3213, Z -5.5000, A 0.000, B 0.000, C 0.000 }
gfCNCPoint4[15177] = {X 419.8632, Y 96.5017, Z -5.5000, A 0.000, B 0.000, C 0.000 }
gfCNCPoint4[15178] = {X 419.8667, Y 97.0654, Z -5.5000, A 0.000, B 0.000, C 0.000 }
gfCNCPoint4[15179] = {X 419.8667, Y 98.0000, Z -5.5000, A 0.000, B 0.000, C 0.000 }
gfCNCPoint4[15180] = {X 419.7624, Y 98.9257, Z -5.5000, A 0.000, B 0.000, C 0.000 }
gfCNCPoint4[15181] = {X 419.4547, Y 99.8050, Z -5.5000, A 0.000, B 0.000, C 0.000 }
gfCNCPoint4[15182] = {X 418.9591, Y 100.5937, Z -5.5000, A 0.000, B 0.000, C 0.000 }
gfCNCPoint4[15183] = {X 418.3004, Y 101.2524, Z -5.5000, A 0.000, B 0.000, C 0.000 }
gfCNCPoint4[15184] = {X 417.5117, Y 101.7480, Z -5.5000, A 0.000, B 0.000, C 0.000 }
gfCNCPoint4[15185] = {X 416.6324, Y 102.0557, Z -5.5000, A 0.000, B 0.000, C 0.000 }
gfCNCPoint4[15186] = {X 415.7067, Y 102.1600, Z -5.5000, A 0.000, B 0.000, C 0.000 }
gfCNCPoint4[15187] = {X 396.4059, Y 102.1600, Z -5.5000, A 0.000, B 0.000, C 0.000 }
gfCNCPoint4[15188] = {X 395.4803, Y 102.0557, Z -5.5000, A 0.000, B 0.000, C 0.000 }
gfCNCPoint4[15189] = {X 394.6010, Y 101.7480, Z -5.5000, A 0.000, B 0.000, C 0.000 }
gfCNCPoint4[15190] = {X 393.8122, Y 101.2524, Z -5.5000, A 0.000, B 0.000, C 0.000 }
gfCNCPoint4[15191] = {X 393.1535, Y 100.5937, Z -5.5000, A 0.000, B 0.000, C 0.000 }
gfCNCPoint4[15192] = {X 392.6579, Y 99.8050, Z -5.5000, A 0.000, B 0.000, C 0.000 }
gfCNCPoint4[15193] = {X 392.3502, Y 98.9257, Z -5.5000, A 0.000, B 0.000, C 0.000 }
gfCNCPoint4[15194] = {X 392.2459, Y 98.0000, Z -5.5000, A 0.000, B 0.000, C 0.000 }
gfCNCPoint4[15195] = {X 392.2459, Y 97.0659, Z -5.5000, A 0.000, B 0.000, C 0.000 }
gfCNCPoint4[15196] = {X 392.3508, Y 96.1380, Z -5.5000, A 0.000, B 0.000, C 0.000 }
gfCNCPoint4[15197] = {X 392.6599, Y 95.2568, Z -5.5000, A 0.000, B 0.000, C 0.000 }
gfCNCPoint4[15198] = {X 393.1579, Y 94.4667, Z -5.5000, A 0.000, B 0.000, C 0.000 }
gfCNCPoint4[15199] = {X 393.8195, Y 93.8077, Z -5.5000, A 0.000, B 0.000, C 0.000 }
gfCNCPoint4[15200] = {X 394.6115, Y 93.3129, Z -5.5000, A 0.000, B 0.000, C 0.000 }
gfCNCPoint4[15201] = {X 395.4939, Y 93.0071, Z -5.5000, A 0.000, B 0.000, C 0.000 }
gfCNCPoint4[15202] = {X 396.4223, Y 92.9060, Z -5.5000, A 0.000, B 0.000, C 0.000 }
gfCNCPoint4[15203] = {X 397.3693, Y 92.8625, Z -5.5000, A 0.000, B 0.000, C 0.000 }
gfCNCPoint4[15204] = {X 398.3131, Y 92.7728, Z -5.5000, A 0.000, B 0.000, C 0.000 }
gfCNCPoint4[15205] = {X 398.9990, Y 92.6064, Z -5.5000, A 0.000, B 0.000, C 0.000 }
gfCNCPoint4[15206] = {X 399.6307, Y 92.2915, Z -5.5000, A 0.000, B 0.000, C 0.000 }
gfCNCPoint4[15207] = {X 413.8852, Y 83.1631, Z -5.5000, A 0.000, B 0.000, C 0.000 }
gfCNCPoint4[15208] = {X 411.7281, Y 79.7946, Z -5.5000, A 0.000, B 0.000, C 0.000 }
gfCNCPoint4[15209] = {X 413.9284, Y 83.2305, Z -5.5000, A 0.000, B 0.000, C 0.000 }
gfCNCPoint4[15210] = {X 428.5798, Y 73.8480, Z -5.5000, A 0.000, B 0.000, C 0.000 }
gfCNCPoint4[15211] = {X 403.8433, Y 64.1428, Z -5.5000, A 0.000, B 0.000, C 0.000 }
gfCNCPoint4[15212] = {X 402.1208, Y 63.5727, Z -5.5000, A 0.000, B 0.000, C 0.000 }
gfCNCPoint4[15213] = {X 400.3462, Y 63.1949, Z -5.5000, A 0.000, B 0.000, C 0.000 }
gfCNCPoint4[15214] = {X 398.5408, Y 63.0140, Z -5.5000, A 0.000, B 0.000, C 0.000 }
gfCNCPoint4[15215] = {X 397.6404, Y 62.9096, Z -5.5000, A 0.000, B 0.000, C 0.000 }
gfCNCPoint4[15216] = {X 396.7853, Y 62.6090, Z -5.5000, A 0.000, B 0.000, C 0.000 }
gfCNCPoint4[15217] = {X 396.0177, Y 62.1269, Z -5.5000, A 0.000, B 0.000, C 0.000 }
gfCNCPoint4[15218] = {X 395.3754, Y 61.4874, Z -5.5000, A 0.000, B 0.000, C 0.000 }
gfCNCPoint4[15219] = {X 394.8902, Y 60.7217, Z -5.5000, A 0.000, B 0.000, C 0.000 }
gfCNCPoint4[15220] = {X 394.5860, Y 59.8679, Z -5.5000, A 0.000, B 0.000, C 0.000 }
gfCNCPoint4[15221] = {X 394.4779, Y 58.9680, Z -5.5000, A 0.000, B 0.000, C 0.000 }
gfCNCPoint4[15222] = {X 394.4777, Y 58.0000, Z -5.5000, A 0.000, B 0.000, C 0.000 }
gfCNCPoint4[15223] = {X 394.5800, Y 57.0921, Z -5.5000, A 0.000, B 0.000, C 0.000 }
gfCNCPoint4[15224] = {X 394.8818, Y 56.2298, Z -5.5000, A 0.000, B 0.000, C 0.000 }
gfCNCPoint4[15225] = {X 395.3678, Y 55.4562, Z -5.5000, A 0.000, B 0.000, C 0.000 }
gfCNCPoint4[15226] = {X 396.0139, Y 54.8101, Z -5.5000, A 0.000, B 0.000, C 0.000 }
gfCNCPoint4[15227] = {X 396.7875, Y 54.3240, Z -5.5000, A 0.000, B 0.000, C 0.000 }
gfCNCPoint4[15228] = {X 397.6498, Y 54.0223, Z -5.5000, A 0.000, B 0.000, C 0.000 }
gfCNCPoint4[15229] = {X 398.5577, Y 53.9200, Z -5.5000, A 0.000, B 0.000, C 0.000 }
gfCNCPoint4[15230] = {X 419.4886, Y 53.9200, Z -5.5000, A 0.000, B 0.000, C 0.000 }
gfCNCPoint4[15231] = {X 420.3965, Y 54.0223, Z -5.5000, A 0.000, B 0.000, C 0.000 }
gfCNCPoint4[15232] = {X 421.2589, Y 54.3240, Z -5.5000, A 0.000, B 0.000, C 0.000 }
gfCNCPoint4[15233] = {X 422.0324, Y 54.8101, Z -5.5000, A 0.000, B 0.000, C 0.000 }
gfCNCPoint4[15234] = {X 422.6785, Y 55.4562, Z -5.5000, A 0.000, B 0.000, C 0.000 }
gfCNCPoint4[15235] = {X 423.1646, Y 56.2298, Z -5.5000, A 0.000, B 0.000, C 0.000 }
gfCNCPoint4[15236] = {X 423.4663, Y 57.0921, Z -5.5000, A 0.000, B 0.000, C 0.000 }
gfCNCPoint4[15237] = {X 423.5686, Y 58.0000, Z -5.5000, A 0.000, B 0.000, C 0.000 }
gfCNCPoint4[15238] = {X 423.5686, Y 58.3960, Z -5.5000, A 0.000, B 0.000, C 0.000 }
gfCNCPoint4[15239] = {X 429.5238, Y 60.7164, Z -5.5000, A 0.000, B 0.000, C 0.000 }
gfCNCPoint4[15240] = {X 458.0983, Y 72.0537, Z -5.5000, A 0.000, B 0.000, C 0.000 }
gfCNCPoint4[15241] = {X 458.1006, Y 62.9982, Z -5.5000, A 0.000, B 0.000, C 0.000 }
gfCNCPoint4[15242] = {X 457.9642, Y 62.9839, Z -5.5000, A 0.000, B 0.000, C 0.000 }
gfCNCPoint4[15243] = {X 457.8283, Y 62.9649, Z -5.5000, A 0.000, B 0.000, C 0.000 }
gfCNCPoint4[15244] = {X 456.9089, Y 62.7079, Z -5.5000, A 0.000, B 0.000, C 0.000 }
gfCNCPoint4[15245] = {X 456.0743, Y 62.2442, Z -5.5000, A 0.000, B 0.000, C 0.000 }
gfCNCPoint4[15246] = {X 455.3704, Y 61.5993, Z -5.5000, A 0.000, B 0.000, C 0.000 }
gfCNCPoint4[15247] = {X 454.8356, Y 60.8084, Z -5.5000, A 0.000, B 0.000, C 0.000 }
gfCNCPoint4[15248] = {X 454.4993, Y 59.9149, Z -5.5000, A 0.000, B 0.000, C 0.000 }
gfCNCPoint4[15249] = {X 454.3797, Y 58.9678, Z -5.5000, A 0.000, B 0.000, C 0.000 }
gfCNCPoint4[15250] = {X 454.3796, Y 58.0000, Z -5.5000, A 0.000, B 0.000, C 0.000 }
gfCNCPoint4[15251] = {X 454.4819, Y 57.0921, Z -5.5000, A 0.000, B 0.000, C 0.000 }
gfCNCPoint4[15252] = {X 454.7837, Y 56.2298, Z -5.5000, A 0.000, B 0.000, C 0.000 }
gfCNCPoint4[15253] = {X 455.2697, Y 55.4562, Z -5.5000, A 0.000, B 0.000, C 0.000 }
gfCNCPoint4[15254] = {X 455.9158, Y 54.8101, Z -5.5000, A 0.000, B 0.000, C 0.000 }
gfCNCPoint4[15255] = {X 456.6894, Y 54.3240, Z -5.5000, A 0.000, B 0.000, C 0.000 }
gfCNCPoint4[15256] = {X 457.5517, Y 54.0223, Z -5.5000, A 0.000, B 0.000, C 0.000 }
gfCNCPoint4[15257] = {X 458.4596, Y 53.9200, Z -5.5000, A 0.000, B 0.000, C 0.000 }
gfCNCPoint4[15258] = {X 475.0000, Y 53.9200, Z -5.5000, A 0.000, B 0.000, C 0.000 }
gfCNCPoint4[15259] = {X 475.9079, Y 54.0223, Z -5.5000, A 0.000, B 0.000, C 0.000 }
gfCNCPoint4[15260] = {X 476.7702, Y 54.3240, Z -5.5000, A 0.000, B 0.000, C 0.000 }
gfCNCPoint4[15261] = {X 477.5438, Y 54.8101, Z -5.5000, A 0.000, B 0.000, C 0.000 }
gfCNCPoint4[15262] = {X 478.1899, Y 55.4562, Z -5.5000, A 0.000, B 0.000, C 0.000 }
gfCNCPoint4[15263] = {X 478.6760, Y 56.2298, Z -5.5000, A 0.000, B 0.000, C 0.000 }
gfCNCPoint4[15264] = {X 478.9777, Y 57.0921, Z -5.5000, A 0.000, B 0.000, C 0.000 }
gfCNCPoint4[15265] = {X 479.0800, Y 58.0000, Z -5.5000, A 0.000, B 0.000, C 0.000 }
gfCNCPoint4[15266] = {X 479.0800, Y 58.9342, Z -5.5000, A 0.000, B 0.000, C 0.000 }
gfCNCPoint4[15267] = {X 478.9888, Y 59.7917, Z -5.5000, A 0.000, B 0.000, C 0.000 }
gfCNCPoint4[15268] = {X 478.7195, Y 60.6109, Z -5.5000, A 0.000, B 0.000, C 0.000 }
gfCNCPoint4[15269] = {X 478.2840, Y 61.3552, Z -5.5000, A 0.000, B 0.000, C 0.000 }
gfCNCPoint4[15270] = {X 477.7017, Y 61.9914, Z -5.5000, A 0.000, B 0.000, C 0.000 }
gfCNCPoint4[15271] = {X 476.9988, Y 62.4909, Z -5.5000, A 0.000, B 0.000, C 0.000 }
gfCNCPoint4[15272] = {X 476.2066, Y 62.8316, Z -5.5000, A 0.000, B 0.000, C 0.000 }
gfCNCPoint4[15273] = {X 475.3605, Y 62.9981, Z -5.5000, A 0.000, B 0.000, C 0.000 }
gfCNCPoint4[15274] = {X 475.3609, Y 92.9628, Z -5.5000, A 0.000, B 0.000, C 0.000 }
gfCNCPoint4[15275] = {X 475.8409, Y 93.0732, Z -5.5000, A 0.000, B 0.000, C 0.000 }
gfCNCPoint4[15276] = {X 476.3128, Y 93.2143, Z -5.5000, A 0.000, B 0.000, C 0.000 }
gfCNCPoint4[15277] = {X 477.0788, Y 93.5626, Z -5.5000, A 0.000, B 0.000, C 0.000 }
gfCNCPoint4[15278] = {X 477.7563, Y 94.0615, Z -5.5000, A 0.000, B 0.000, C 0.000 }
gfCNCPoint4[15279] = {X 478.3162, Y 94.6896, Z -5.5000, A 0.000, B 0.000, C 0.000 }
gfCNCPoint4[15280] = {X 478.7343, Y 95.4198, Z -5.5000, A 0.000, B 0.000, C 0.000 }
gfCNCPoint4[15281] = {X 478.9926, Y 96.2206, Z -5.5000, A 0.000, B 0.000, C 0.000 }
gfCNCPoint4[15282] = {X 479.0800, Y 97.0575, Z -5.5000, A 0.000, B 0.000, C 0.000 }
gfCNCPoint4[15283] = {X 479.0800, Y 98.0000, Z -5.5000, A 0.000, B 0.000, C 0.000 }
gfCNCPoint4[15284] = {X 478.9777, Y 98.9079, Z -5.5000, A 0.000, B 0.000, C 0.000 }
gfCNCPoint4[15285] = {X 478.6760, Y 99.7702, Z -5.5000, A 0.000, B 0.000, C 0.000 }
gfCNCPoint4[15286] = {X 478.1899, Y 100.5438, Z -5.5000, A 0.000, B 0.000, C 0.000 }
gfCNCPoint4[15287] = {X 477.5438, Y 101.1899, Z -5.5000, A 0.000, B 0.000, C 0.000 }
gfCNCPoint4[15288] = {X 476.7702, Y 101.6760, Z -5.5000, A 0.000, B 0.000, C 0.000 }
gfCNCPoint4[15289] = {X 475.9079, Y 101.9777, Z -5.5000, A 0.000, B 0.000, C 0.000 }
gfCNCPoint4[15290] = {X 475.0000, Y 102.0800, Z -5.5000, A 0.000, B 0.000, C 0.000 }
gfCNCPoint4[15291] = {X 458.4596, Y 102.0800, Z -5.5000, A 0.000, B 0.000, C 0.000 }
gfCNCPoint4[15292] = {X 457.5517, Y 101.9777, Z -5.5000, A 0.000, B 0.000, C 0.000 }
gfCNCPoint4[15293] = {X 456.6894, Y 101.6760, Z -5.5000, A 0.000, B 0.000, C 0.000 }
gfCNCPoint4[15294] = {X 455.9158, Y 101.1899, Z -5.5000, A 0.000, B 0.000, C 0.000 }
gfCNCPoint4[15295] = {X 455.2697, Y 100.5438, Z -5.5000, A 0.000, B 0.000, C 0.000 }
gfCNCPoint4[15296] = {X 454.7837, Y 99.7702, Z -5.5000, A 0.000, B 0.000, C 0.000 }
gfCNCPoint4[15297] = {X 454.4819, Y 98.9079, Z -5.5000, A 0.000, B 0.000, C 0.000 }
gfCNCPoint4[15298] = {X 454.3796, Y 98.0000, Z -5.5000, A 0.000, B 0.000, C 0.000 }
gfCNCPoint4[15299] = {X 454.3796, Y 97.0659, Z -5.5000, A 0.000, B 0.000, C 0.000 }
gfCNCPoint4[15300] = {X 454.4707, Y 96.2088, Z -5.5000, A 0.000, B 0.000, C 0.000 }
gfCNCPoint4[15301] = {X 454.7398, Y 95.3899, Z -5.5000, A 0.000, B 0.000, C 0.000 }
gfCNCPoint4[15302] = {X 455.1749, Y 94.6458, Z -5.5000, A 0.000, B 0.000, C 0.000 }
gfCNCPoint4[15303] = {X 455.7566, Y 94.0098, Z -5.5000, A 0.000, B 0.000, C 0.000 }
gfCNCPoint4[15304] = {X 456.4590, Y 93.5101, Z -5.5000, A 0.000, B 0.000, C 0.000 }
gfCNCPoint4[15305] = {X 457.2507, Y 93.1692, Z -5.5000, A 0.000, B 0.000, C 0.000 }
gfCNCPoint4[15306] = {X 458.0963, Y 93.0021, Z -5.5000, A 0.000, B 0.000, C 0.000 }
gfCNCPoint4[15307] = {X 458.0963, Y 85.4313, Z -5.5000, A 0.000, B 0.000, C 0.000 }
gfCNCPoint4[15308] = {X 444.8324, Y 80.2318, Z -5.5000, A 0.000, B 0.000, C 0.000 }
gfCNCPoint4[15309] = {X 419.7829, Y 96.4584, Z -5.5000, A 0.000, B 0.000, C 0.000 }
gfCNCPoint4[15310] = {X 419.7867, Y 97.0657, Z -5.5000, A 0.000, B 0.000, C 0.000 }
gfCNCPoint4[15311] = {X 419.7867, Y 98.0000, Z -5.5000, A 0.000, B 0.000, C 0.000 }
gfCNCPoint4[15312] = {X 419.6844, Y 98.9079, Z -5.5000, A 0.000, B 0.000, C 0.000 }
gfCNCPoint4[15313] = {X 419.3827, Y 99.7702, Z -5.5000, A 0.000, B 0.000, C 0.000 }
gfCNCPoint4[15314] = {X 418.8966, Y 100.5438, Z -5.5000, A 0.000, B 0.000, C 0.000 }
gfCNCPoint4[15315] = {X 418.2505, Y 101.1899, Z -5.5000, A 0.000, B 0.000, C 0.000 }
gfCNCPoint4[15316] = {X 417.4769, Y 101.6760, Z -5.5000, A 0.000, B 0.000, C 0.000 }
gfCNCPoint4[15317] = {X 416.6146, Y 101.9777, Z -5.5000, A 0.000, B 0.000, C 0.000 }
gfCNCPoint4[15318] = {X 415.7067, Y 102.0800, Z -5.5000, A 0.000, B 0.000, C 0.000 }
gfCNCPoint4[15319] = {X 396.4059, Y 102.0800, Z -5.5000, A 0.000, B 0.000, C 0.000 }
gfCNCPoint4[15320] = {X 395.4981, Y 101.9777, Z -5.5000, A 0.000, B 0.000, C 0.000 }
gfCNCPoint4[15321] = {X 394.6357, Y 101.6760, Z -5.5000, A 0.000, B 0.000, C 0.000 }
gfCNCPoint4[15322] = {X 393.8621, Y 101.1899, Z -5.5000, A 0.000, B 0.000, C 0.000 }
gfCNCPoint4[15323] = {X 393.2161, Y 100.5438, Z -5.5000, A 0.000, B 0.000, C 0.000 }
gfCNCPoint4[15324] = {X 392.7300, Y 99.7702, Z -5.5000, A 0.000, B 0.000, C 0.000 }
gfCNCPoint4[15325] = {X 392.4282, Y 98.9079, Z -5.5000, A 0.000, B 0.000, C 0.000 }
gfCNCPoint4[15326] = {X 392.3259, Y 98.0000, Z -5.5000, A 0.000, B 0.000, C 0.000 }
gfCNCPoint4[15327] = {X 392.3259, Y 97.0659, Z -5.5000, A 0.000, B 0.000, C 0.000 }
gfCNCPoint4[15328] = {X 392.4288, Y 96.1557, Z -5.5000, A 0.000, B 0.000, C 0.000 }
gfCNCPoint4[15329] = {X 392.7321, Y 95.2913, Z -5.5000, A 0.000, B 0.000, C 0.000 }
gfCNCPoint4[15330] = {X 393.2206, Y 94.5164, Z -5.5000, A 0.000, B 0.000, C 0.000 }
gfCNCPoint4[15331] = {X 393.8697, Y 93.8700, Z -5.5000, A 0.000, B 0.000, C 0.000 }
gfCNCPoint4[15332] = {X 394.6467, Y 93.3847, Z -5.5000, A 0.000, B 0.000, C 0.000 }
gfCNCPoint4[15333] = {X 395.5123, Y 93.0850, Z -5.5000, A 0.000, B 0.000, C 0.000 }
gfCNCPoint4[15334] = {X 396.4230, Y 92.9860, Z -5.5000, A 0.000, B 0.000, C 0.000 }
gfCNCPoint4[15335] = {X 397.3746, Y 92.9424, Z -5.5000, A 0.000, B 0.000, C 0.000 }
gfCNCPoint4[15336] = {X 398.3229, Y 92.8522, Z -5.5000, A 0.000, B 0.000, C 0.000 }
gfCNCPoint4[15337] = {X 399.0264, Y 92.6816, Z -5.5000, A 0.000, B 0.000, C 0.000 }
gfCNCPoint4[15338] = {X 399.6742, Y 92.3587, Z -5.5000, A 0.000, B 0.000, C 0.000 }
gfCNCPoint4[15339] = {X 413.9284, Y 83.2305, Z -5.5000, A 0.000, B 0.000, C 0.000 }
gfCNCPoint4[15340] = {X 411.7648, Y 79.8520, Z -5.5000, A 0.000, B 0.000, C 0.000 }
gfCNCPoint4[15341] = {X 411.7671, Y 79.8505, Z -5.5000, A 0.000, B 0.000, C 0.000 }
gfCNCPoint4[15342] = {X 413.9651, Y 83.2879, Z -5.5000, A 0.000, B 0.000, C 0.000 }
gfCNCPoint4[15343] = {X 428.7551, Y 73.8308, Z -5.5000, A 0.000, B 0.000, C 0.000 }
gfCNCPoint4[15344] = {X 403.8726, Y 64.0684, Z -5.5000, A 0.000, B 0.000, C 0.000 }
gfCNCPoint4[15345] = {X 402.1412, Y 63.4953, Z -5.5000, A 0.000, B 0.000, C 0.000 }
gfCNCPoint4[15346] = {X 400.3574, Y 63.1157, Z -5.5000, A 0.000, B 0.000, C 0.000 }
gfCNCPoint4[15347] = {X 398.5427, Y 62.9340, Z -5.5000, A 0.000, B 0.000, C 0.000 }
gfCNCPoint4[15348] = {X 397.6551, Y 62.8309, Z -5.5000, A 0.000, B 0.000, C 0.000 }
gfCNCPoint4[15349] = {X 396.8125, Y 62.5333, Z -5.5000, A 0.000, B 0.000, C 0.000 }
gfCNCPoint4[15350] = {X 396.0571, Y 62.0560, Z -5.5000, A 0.000, B 0.000, C 0.000 }
gfCNCPoint4[15351] = {X 395.4264, Y 61.4230, Z -5.5000, A 0.000, B 0.000, C 0.000 }
gfCNCPoint4[15352] = {X 394.9520, Y 60.6657, Z -5.5000, A 0.000, B 0.000, C 0.000 }
gfCNCPoint4[15353] = {X 394.6575, Y 59.8220, Z -5.5000, A 0.000, B 0.000, C 0.000 }
gfCNCPoint4[15354] = {X 394.5577, Y 58.9341, Z -5.5000, A 0.000, B 0.000, C 0.000 }
gfCNCPoint4[15355] = {X 394.5577, Y 58.0000, Z -5.5000, A 0.000, B 0.000, C 0.000 }
gfCNCPoint4[15356] = {X 394.6580, Y 57.1099, Z -5.5000, A 0.000, B 0.000, C 0.000 }
gfCNCPoint4[15357] = {X 394.9538, Y 56.2645, Z -5.5000, A 0.000, B 0.000, C 0.000 }
gfCNCPoint4[15358] = {X 395.4304, Y 55.5060, Z -5.5000, A 0.000, B 0.000, C 0.000 }
gfCNCPoint4[15359] = {X 396.0638, Y 54.8727, Z -5.5000, A 0.000, B 0.000, C 0.000 }
gfCNCPoint4[15360] = {X 396.8222, Y 54.3961, Z -5.5000, A 0.000, B 0.000, C 0.000 }
gfCNCPoint4[15361] = {X 397.6676, Y 54.1003, Z -5.5000, A 0.000, B 0.000, C 0.000 }
gfCNCPoint4[15362] = {X 398.5577, Y 54.0000, Z -5.5000, A 0.000, B 0.000, C 0.000 }
gfCNCPoint4[15363] = {X 419.4886, Y 54.0000, Z -5.5000, A 0.000, B 0.000, C 0.000 }
gfCNCPoint4[15364] = {X 420.3787, Y 54.1003, Z -5.5000, A 0.000, B 0.000, C 0.000 }
gfCNCPoint4[15365] = {X 421.2241, Y 54.3961, Z -5.5000, A 0.000, B 0.000, C 0.000 }
gfCNCPoint4[15366] = {X 421.9826, Y 54.8727, Z -5.5000, A 0.000, B 0.000, C 0.000 }
gfCNCPoint4[15367] = {X 422.6159, Y 55.5060, Z -5.5000, A 0.000, B 0.000, C 0.000 }
gfCNCPoint4[15368] = {X 423.0925, Y 56.2645, Z -5.5000, A 0.000, B 0.000, C 0.000 }
gfCNCPoint4[15369] = {X 423.3883, Y 57.1099, Z -5.5000, A 0.000, B 0.000, C 0.000 }
gfCNCPoint4[15370] = {X 423.4886, Y 58.0000, Z -5.5000, A 0.000, B 0.000, C 0.000 }
gfCNCPoint4[15371] = {X 423.4886, Y 58.4507, Z -5.5000, A 0.000, B 0.000, C 0.000 }
gfCNCPoint4[15372] = {X 429.4945, Y 60.7908, Z -5.5000, A 0.000, B 0.000, C 0.000 }
gfCNCPoint4[15373] = {X 458.1783, Y 72.1715, Z -5.5000, A 0.000, B 0.000, C 0.000 }
gfCNCPoint4[15374] = {X 458.1788, Y 63.0389, Z -5.5000, A 0.000, B 0.000, C 0.000 }
gfCNCPoint4[15375] = {X 458.1841, Y 62.9246, Z -5.5000, A 0.000, B 0.000, C 0.000 }
gfCNCPoint4[15376] = {X 458.0120, Y 62.9089, Z -5.5000, A 0.000, B 0.000, C 0.000 }
gfCNCPoint4[15377] = {X 457.8407, Y 62.8859, Z -5.5000, A 0.000, B 0.000, C 0.000 }
gfCNCPoint4[15378] = {X 456.9342, Y 62.6318, Z -5.5000, A 0.000, B 0.000, C 0.000 }
gfCNCPoint4[15379] = {X 456.1122, Y 62.1728, Z -5.5000, A 0.000, B 0.000, C 0.000 }
gfCNCPoint4[15380] = {X 455.4202, Y 61.5345, Z -5.5000, A 0.000, B 0.000, C 0.000 }
gfCNCPoint4[15381] = {X 454.8966, Y 60.7521, Z -5.5000, A 0.000, B 0.000, C 0.000 }
gfCNCPoint4[15382] = {X 454.5704, Y 59.8690, Z -5.5000, A 0.000, B 0.000, C 0.000 }
gfCNCPoint4[15383] = {X 454.4596, Y 58.9341, Z -5.5000, A 0.000, B 0.000, C 0.000 }
gfCNCPoint4[15384] = {X 454.4596, Y 58.0000, Z -5.5000, A 0.000, B 0.000, C 0.000 }
gfCNCPoint4[15385] = {X 454.5599, Y 57.1099, Z -5.5000, A 0.000, B 0.000, C 0.000 }
gfCNCPoint4[15386] = {X 454.8557, Y 56.2645, Z -5.5000, A 0.000, B 0.000, C 0.000 }
gfCNCPoint4[15387] = {X 455.3323, Y 55.5060, Z -5.5000, A 0.000, B 0.000, C 0.000 }
gfCNCPoint4[15388] = {X 455.9656, Y 54.8727, Z -5.5000, A 0.000, B 0.000, C 0.000 }
gfCNCPoint4[15389] = {X 456.7241, Y 54.3961, Z -5.5000, A 0.000, B 0.000, C 0.000 }
gfCNCPoint4[15390] = {X 457.5695, Y 54.1003, Z -5.5000, A 0.000, B 0.000, C 0.000 }
gfCNCPoint4[15391] = {X 458.4596, Y 54.0000, Z -5.5000, A 0.000, B 0.000, C 0.000 }
gfCNCPoint4[15392] = {X 475.0000, Y 54.0000, Z -5.5000, A 0.000, B 0.000, C 0.000 }
gfCNCPoint4[15393] = {X 475.8901, Y 54.1003, Z -5.5000, A 0.000, B 0.000, C 0.000 }
gfCNCPoint4[15394] = {X 476.7355, Y 54.3961, Z -5.5000, A 0.000, B 0.000, C 0.000 }
gfCNCPoint4[15395] = {X 477.4940, Y 54.8727, Z -5.5000, A 0.000, B 0.000, C 0.000 }
gfCNCPoint4[15396] = {X 478.1273, Y 55.5060, Z -5.5000, A 0.000, B 0.000, C 0.000 }
gfCNCPoint4[15397] = {X 478.6039, Y 56.2645, Z -5.5000, A 0.000, B 0.000, C 0.000 }
gfCNCPoint4[15398] = {X 478.8997, Y 57.1099, Z -5.5000, A 0.000, B 0.000, C 0.000 }
gfCNCPoint4[15399] = {X 479.0000, Y 58.0000, Z -5.5000, A 0.000, B 0.000, C 0.000 }
gfCNCPoint4[15400] = {X 478.9999, Y 58.9671, Z -5.5000, A 0.000, B 0.000, C 0.000 }
gfCNCPoint4[15401] = {X 478.9023, Y 59.8127, Z -5.5000, A 0.000, B 0.000, C 0.000 }
gfCNCPoint4[15402] = {X 478.6281, Y 60.6184, Z -5.5000, A 0.000, B 0.000, C 0.000 }
gfCNCPoint4[15403] = {X 478.1896, Y 61.3479, Z -5.5000, A 0.000, B 0.000, C 0.000 }
gfCNCPoint4[15404] = {X 477.6066, Y 61.9681, Z -5.5000, A 0.000, B 0.000, C 0.000 }
gfCNCPoint4[15405] = {X 476.9056, Y 62.4510, Z -5.5000, A 0.000, B 0.000, C 0.000 }
gfCNCPoint4[15406] = {X 476.1184, Y 62.7745, Z -5.5000, A 0.000, B 0.000, C 0.000 }
gfCNCPoint4[15407] = {X 475.2805, Y 62.9242, Z -5.5000, A 0.000, B 0.000, C 0.000 }
gfCNCPoint4[15408] = {X 475.2809, Y 93.0289, Z -5.5000, A 0.000, B 0.000, C 0.000 }
gfCNCPoint4[15409] = {X 475.7887, Y 93.1422, Z -5.5000, A 0.000, B 0.000, C 0.000 }
gfCNCPoint4[15410] = {X 476.2874, Y 93.2902, Z -5.5000, A 0.000, B 0.000, C 0.000 }
gfCNCPoint4[15411] = {X 477.0383, Y 93.6316, Z -5.5000, A 0.000, B 0.000, C 0.000 }
gfCNCPoint4[15412] = {X 477.7025, Y 94.1207, Z -5.5000, A 0.000, B 0.000, C 0.000 }
gfCNCPoint4[15413] = {X 478.2513, Y 94.7364, Z -5.5000, A 0.000, B 0.000, C 0.000 }
gfCNCPoint4[15414] = {X 478.6612, Y 95.4521, Z -5.5000, A 0.000, B 0.000, C 0.000 }
gfCNCPoint4[15415] = {X 478.9144, Y 96.2371, Z -5.5000, A 0.000, B 0.000, C 0.000 }
gfCNCPoint4[15416] = {X 479.0000, Y 97.0575, Z -5.5000, A 0.000, B 0.000, C 0.000 }
gfCNCPoint4[15417] = {X 479.0000, Y 98.0000, Z -5.5000, A 0.000, B 0.000, C 0.000 }
gfCNCPoint4[15418] = {X 478.8997, Y 98.8901, Z -5.5000, A 0.000, B 0.000, C 0.000 }
gfCNCPoint4[15419] = {X 478.6039, Y 99.7355, Z -5.5000, A 0.000, B 0.000, C 0.000 }
gfCNCPoint4[15420] = {X 478.1273, Y 100.4940, Z -5.5000, A 0.000, B 0.000, C 0.000 }
gfCNCPoint4[15421] = {X 477.4940, Y 101.1273, Z -5.5000, A 0.000, B 0.000, C 0.000 }
gfCNCPoint4[15422] = {X 476.7355, Y 101.6039, Z -5.5000, A 0.000, B 0.000, C 0.000 }
gfCNCPoint4[15423] = {X 475.8901, Y 101.8997, Z -5.5000, A 0.000, B 0.000, C 0.000 }
gfCNCPoint4[15424] = {X 475.0000, Y 102.0000, Z -5.5000, A 0.000, B 0.000, C 0.000 }
gfCNCPoint4[15425] = {X 458.4596, Y 102.0000, Z -5.5000, A 0.000, B 0.000, C 0.000 }
gfCNCPoint4[15426] = {X 457.5695, Y 101.8997, Z -5.5000, A 0.000, B 0.000, C 0.000 }
gfCNCPoint4[15427] = {X 456.7241, Y 101.6039, Z -5.5000, A 0.000, B 0.000, C 0.000 }
gfCNCPoint4[15428] = {X 455.9656, Y 101.1273, Z -5.5000, A 0.000, B 0.000, C 0.000 }
gfCNCPoint4[15429] = {X 455.3323, Y 100.4940, Z -5.5000, A 0.000, B 0.000, C 0.000 }
gfCNCPoint4[15430] = {X 454.8557, Y 99.7355, Z -5.5000, A 0.000, B 0.000, C 0.000 }
gfCNCPoint4[15431] = {X 454.5599, Y 98.8901, Z -5.5000, A 0.000, B 0.000, C 0.000 }
gfCNCPoint4[15432] = {X 454.4596, Y 98.0000, Z -5.5000, A 0.000, B 0.000, C 0.000 }
gfCNCPoint4[15433] = {X 454.4596, Y 97.0659, Z -5.5000, A 0.000, B 0.000, C 0.000 }
gfCNCPoint4[15434] = {X 454.5511, Y 96.2154, Z -5.5000, A 0.000, B 0.000, C 0.000 }
gfCNCPoint4[15435] = {X 454.8213, Y 95.4037, Z -5.5000, A 0.000, B 0.000, C 0.000 }
gfCNCPoint4[15436] = {X 455.2580, Y 94.6681, Z -5.5000, A 0.000, B 0.000, C 0.000 }
gfCNCPoint4[15437] = {X 455.8411, Y 94.0422, Z -5.5000, A 0.000, B 0.000, C 0.000 }
gfCNCPoint4[15438] = {X 456.5439, Y 93.5545, Z -5.5000, A 0.000, B 0.000, C 0.000 }
gfCNCPoint4[15439] = {X 457.3344, Y 93.2275, Z -5.5000, A 0.000, B 0.000, C 0.000 }
gfCNCPoint4[15440] = {X 458.1763, Y 93.0760, Z -5.5000, A 0.000, B 0.000, C 0.000 }
gfCNCPoint4[15441] = {X 458.1763, Y 85.3767, Z -5.5000, A 0.000, B 0.000, C 0.000 }
gfCNCPoint4[15442] = {X 445.0145, Y 80.2173, Z -5.5000, A 0.000, B 0.000, C 0.000 }
gfCNCPoint4[15443] = {X 444.8242, Y 80.1418, Z -5.5000, A 0.000, B 0.000, C 0.000 }
gfCNCPoint4[15444] = {X 419.7026, Y 96.4151, Z -5.5000, A 0.000, B 0.000, C 0.000 }
gfCNCPoint4[15445] = {X 419.7067, Y 97.0659, Z -5.5000, A 0.000, B 0.000, C 0.000 }
gfCNCPoint4[15446] = {X 419.7067, Y 98.0000, Z -5.5000, A 0.000, B 0.000, C 0.000 }
gfCNCPoint4[15447] = {X 419.6064, Y 98.8901, Z -5.5000, A 0.000, B 0.000, C 0.000 }
gfCNCPoint4[15448] = {X 419.3106, Y 99.7355, Z -5.5000, A 0.000, B 0.000, C 0.000 }
gfCNCPoint4[15449] = {X 418.8340, Y 100.4940, Z -5.5000, A 0.000, B 0.000, C 0.000 }
gfCNCPoint4[15450] = {X 418.2007, Y 101.1273, Z -5.5000, A 0.000, B 0.000, C 0.000 }
gfCNCPoint4[15451] = {X 417.4422, Y 101.6039, Z -5.5000, A 0.000, B 0.000, C 0.000 }
gfCNCPoint4[15452] = {X 416.5968, Y 101.8997, Z -5.5000, A 0.000, B 0.000, C 0.000 }
gfCNCPoint4[15453] = {X 415.7067, Y 102.0000, Z -5.5000, A 0.000, B 0.000, C 0.000 }
gfCNCPoint4[15454] = {X 396.4059, Y 102.0000, Z -5.5000, A 0.000, B 0.000, C 0.000 }
gfCNCPoint4[15455] = {X 395.5159, Y 101.8997, Z -5.5000, A 0.000, B 0.000, C 0.000 }
gfCNCPoint4[15456] = {X 394.6704, Y 101.6039, Z -5.5000, A 0.000, B 0.000, C 0.000 }
gfCNCPoint4[15457] = {X 393.9120, Y 101.1273, Z -5.5000, A 0.000, B 0.000, C 0.000 }
gfCNCPoint4[15458] = {X 393.2786, Y 100.4940, Z -5.5000, A 0.000, B 0.000, C 0.000 }
gfCNCPoint4[15459] = {X 392.8021, Y 99.7355, Z -5.5000, A 0.000, B 0.000, C 0.000 }
gfCNCPoint4[15460] = {X 392.5062, Y 98.8901, Z -5.5000, A 0.000, B 0.000, C 0.000 }
gfCNCPoint4[15461] = {X 392.4059, Y 98.0000, Z -5.5000, A 0.000, B 0.000, C 0.000 }
gfCNCPoint4[15462] = {X 392.4059, Y 97.0659, Z -5.5000, A 0.000, B 0.000, C 0.000 }
gfCNCPoint4[15463] = {X 392.5068, Y 96.1734, Z -5.5000, A 0.000, B 0.000, C 0.000 }
gfCNCPoint4[15464] = {X 392.8043, Y 95.3258, Z -5.5000, A 0.000, B 0.000, C 0.000 }
gfCNCPoint4[15465] = {X 393.2834, Y 94.5660, Z -5.5000, A 0.000, B 0.000, C 0.000 }
gfCNCPoint4[15466] = {X 393.9199, Y 93.9323, Z -5.5000, A 0.000, B 0.000, C 0.000 }
gfCNCPoint4[15467] = {X 394.6818, Y 93.4566, Z -5.5000, A 0.000, B 0.000, C 0.000 }
gfCNCPoint4[15468] = {X 395.5307, Y 93.1629, Z -5.5000, A 0.000, B 0.000, C 0.000 }
gfCNCPoint4[15469] = {X 396.4237, Y 93.0660, Z -5.5000, A 0.000, B 0.000, C 0.000 }
gfCNCPoint4[15470] = {X 397.3798, Y 93.0222, Z -5.5000, A 0.000, B 0.000, C 0.000 }
gfCNCPoint4[15471] = {X 398.3327, Y 92.9316, Z -5.5000, A 0.000, B 0.000, C 0.000 }
gfCNCPoint4[15472] = {X 399.0537, Y 92.7568, Z -5.5000, A 0.000, B 0.000, C 0.000 }
gfCNCPoint4[15473] = {X 399.7177, Y 92.4258, Z -5.5000, A 0.000, B 0.000, C 0.000 }
gfCNCPoint4[15474] = {X 405.3919, Y 88.7698, Z -5.5000, A 0.000, B 0.000, C 0.000 }
gfCNCPoint4[15475] = {X 413.9651, Y 83.2879, Z -5.5000, A 0.000, B 0.000, C 0.000 }
gfCNCPoint4[15476] = {X 411.7671, Y 79.8505, Z -5.5000, A 0.000, B 0.000, C 0.000 }
gfCNCPoint4[15477] = {X 411.7671, Y 79.8505, Z -2.5000, A 0.000, B 0.000, C 0.000 }
gfCNCPoint4[15478] = {X 411.7671, Y 79.8505, Z 11.0000, A 0.000, B 0.000, C 0.000 }
gfCNCPoint4[15479] = {X 466.3111, Y 28.5934, Z 11.0000, A 0.000, B 0.000, C 0.000 }
gfCNCPoint4[15480] = {X 466.3111, Y 28.5934, Z -2.5000, A 0.000, B 0.000, C 0.000 }
gfCNCPoint4[15481] = {X 466.3111, Y 28.5934, Z -5.5000, A 0.000, B 0.000, C 0.000 }
gfCNCPoint4[15482] = {X 462.2311, Y 28.5935, Z -5.5000, A 0.000, B 0.000, C 0.000 }
gfCNCPoint4[15483] = {X 462.2314, Y 40.9137, Z -5.5000, A 0.000, B 0.000, C 0.000 }
gfCNCPoint4[15484] = {X 462.2399, Y 40.9207, Z -5.5000, A 0.000, B 0.000, C 0.000 }
gfCNCPoint4[15485] = {X 462.8746, Y 41.5911, Z -5.5000, A 0.000, B 0.000, C 0.000 }
gfCNCPoint4[15486] = {X 463.3523, Y 42.3812, Z -5.5000, A 0.000, B 0.000, C 0.000 }
gfCNCPoint4[15487] = {X 463.6513, Y 43.2547, Z -5.5000, A 0.000, B 0.000, C 0.000 }
gfCNCPoint4[15488] = {X 463.7578, Y 44.1718, Z -5.5000, A 0.000, B 0.000, C 0.000 }
gfCNCPoint4[15489] = {X 463.7579, Y 45.0000, Z -5.5000, A 0.000, B 0.000, C 0.000 }
gfCNCPoint4[15490] = {X 463.6496, Y 45.9613, Z -5.5000, A 0.000, B 0.000, C 0.000 }
gfCNCPoint4[15491] = {X 463.3301, Y 46.8744, Z -5.5000, A 0.000, B 0.000, C 0.000 }
gfCNCPoint4[15492] = {X 462.8155, Y 47.6935, Z -5.5000, A 0.000, B 0.000, C 0.000 }
gfCNCPoint4[15493] = {X 462.1314, Y 48.3775, Z -5.5000, A 0.000, B 0.000, C 0.000 }
gfCNCPoint4[15494] = {X 461.3123, Y 48.8922, Z -5.5000, A 0.000, B 0.000, C 0.000 }
gfCNCPoint4[15495] = {X 460.3992, Y 49.2117, Z -5.5000, A 0.000, B 0.000, C 0.000 }
gfCNCPoint4[15496] = {X 459.4379, Y 49.3200, Z -5.5000, A 0.000, B 0.000, C 0.000 }
gfCNCPoint4[15497] = {X 452.9945, Y 49.3200, Z -5.5000, A 0.000, B 0.000, C 0.000 }
gfCNCPoint4[15498] = {X 452.0380, Y 49.2128, Z -5.5000, A 0.000, B 0.000, C 0.000 }
gfCNCPoint4[15499] = {X 451.1291, Y 48.8965, Z -5.5000, A 0.000, B 0.000, C 0.000 }
gfCNCPoint4[15500] = {X 450.3127, Y 48.3868, Z -5.5000, A 0.000, B 0.000, C 0.000 }
gfCNCPoint4[15501] = {X 449.6294, Y 47.7091, Z -5.5000, A 0.000, B 0.000, C 0.000 }
gfCNCPoint4[15502] = {X 449.1132, Y 46.8968, Z -5.5000, A 0.000, B 0.000, C 0.000 }
gfCNCPoint4[15503] = {X 448.7895, Y 45.9905, Z -5.5000, A 0.000, B 0.000, C 0.000 }
gfCNCPoint4[15504] = {X 448.6746, Y 45.0349, Z -5.5000, A 0.000, B 0.000, C 0.000 }
gfCNCPoint4[15505] = {X 448.6749, Y 44.1494, Z -5.5000, A 0.000, B 0.000, C 0.000 }
gfCNCPoint4[15506] = {X 448.7853, Y 43.2364, Z -5.5000, A 0.000, B 0.000, C 0.000 }
gfCNCPoint4[15507] = {X 449.0865, Y 42.3675, Z -5.5000, A 0.000, B 0.000, C 0.000 }
gfCNCPoint4[15508] = {X 449.5648, Y 41.5821, Z -5.5000, A 0.000, B 0.000, C 0.000 }
gfCNCPoint4[15509] = {X 450.1984, Y 40.9157, Z -5.5000, A 0.000, B 0.000, C 0.000 }
gfCNCPoint4[15510] = {X 450.1984, Y 34.4738, Z -5.5000, A 0.000, B 0.000, C 0.000 }
gfCNCPoint4[15511] = {X 447.4750, Y 34.4738, Z -5.5000, A 0.000, B 0.000, C 0.000 }
gfCNCPoint4[15512] = {X 443.1898, Y 42.8171, Z -5.5000, A 0.000, B 0.000, C 0.000 }
gfCNCPoint4[15513] = {X 443.1947, Y 42.8306, Z -5.5000, A 0.000, B 0.000, C 0.000 }
gfCNCPoint4[15514] = {X 443.3605, Y 43.4915, Z -5.5000, A 0.000, B 0.000, C 0.000 }
gfCNCPoint4[15515] = {X 443.4203, Y 44.1703, Z -5.5000, A 0.000, B 0.000, C 0.000 }
gfCNCPoint4[15516] = {X 443.4205, Y 45.0000, Z -5.5000, A 0.000, B 0.000, C 0.000 }
gfCNCPoint4[15517] = {X 443.3122, Y 45.9613, Z -5.5000, A 0.000, B 0.000, C 0.000 }
gfCNCPoint4[15518] = {X 442.9927, Y 46.8744, Z -5.5000, A 0.000, B 0.000, C 0.000 }
gfCNCPoint4[15519] = {X 442.4780, Y 47.6935, Z -5.5000, A 0.000, B 0.000, C 0.000 }
gfCNCPoint4[15520] = {X 441.7939, Y 48.3775, Z -5.5000, A 0.000, B 0.000, C 0.000 }
gfCNCPoint4[15521] = {X 440.9748, Y 48.8922, Z -5.5000, A 0.000, B 0.000, C 0.000 }
gfCNCPoint4[15522] = {X 440.0618, Y 49.2117, Z -5.5000, A 0.000, B 0.000, C 0.000 }
gfCNCPoint4[15523] = {X 439.1005, Y 49.3200, Z -5.5000, A 0.000, B 0.000, C 0.000 }
gfCNCPoint4[15524] = {X 432.5144, Y 49.3200, Z -5.5000, A 0.000, B 0.000, C 0.000 }
gfCNCPoint4[15525] = {X 431.5531, Y 49.2117, Z -5.5000, A 0.000, B 0.000, C 0.000 }
gfCNCPoint4[15526] = {X 430.6401, Y 48.8922, Z -5.5000, A 0.000, B 0.000, C 0.000 }
gfCNCPoint4[15527] = {X 429.8210, Y 48.3775, Z -5.5000, A 0.000, B 0.000, C 0.000 }
gfCNCPoint4[15528] = {X 429.1369, Y 47.6935, Z -5.5000, A 0.000, B 0.000, C 0.000 }
gfCNCPoint4[15529] = {X 428.6223, Y 46.8745, Z -5.5000, A 0.000, B 0.000, C 0.000 }
gfCNCPoint4[15530] = {X 428.3027, Y 45.9614, Z -5.5000, A 0.000, B 0.000, C 0.000 }
gfCNCPoint4[15531] = {X 428.1944, Y 45.0001, Z -5.5000, A 0.000, B 0.000, C 0.000 }
gfCNCPoint4[15532] = {X 428.1948, Y 44.1494, Z -5.5000, A 0.000, B 0.000, C 0.000 }
gfCNCPoint4[15533] = {X 428.2925, Y 43.2935, Z -5.5000, A 0.000, B 0.000, C 0.000 }
gfCNCPoint4[15534] = {X 428.5580, Y 42.4740, Z -5.5000, A 0.000, B 0.000, C 0.000 }
gfCNCPoint4[15535] = {X 428.9809, Y 41.7236, Z -5.5000, A 0.000, B 0.000, C 0.000 }
gfCNCPoint4[15536] = {X 429.5442, Y 41.0719, Z -5.5000, A 0.000, B 0.000, C 0.000 }
gfCNCPoint4[15537] = {X 430.2256, Y 40.5449, Z -5.5000, A 0.000, B 0.000, C 0.000 }
gfCNCPoint4[15538] = {X 430.9981, Y 40.1637, Z -5.5000, A 0.000, B 0.000, C 0.000 }
gfCNCPoint4[15539] = {X 434.9872, Y 32.3554, Z -5.5000, A 0.000, B 0.000, C 0.000 }
gfCNCPoint4[15540] = {X 433.7208, Y 31.4922, Z -5.5000, A 0.000, B 0.000, C 0.000 }
gfCNCPoint4[15541] = {X 432.5819, Y 30.4667, Z -5.5000, A 0.000, B 0.000, C 0.000 }
gfCNCPoint4[15542] = {X 431.5910, Y 29.2976, Z -5.5000, A 0.000, B 0.000, C 0.000 }
gfCNCPoint4[15543] = {X 430.7660, Y 28.0060, Z -5.5000, A 0.000, B 0.000, C 0.000 }
gfCNCPoint4[15544] = {X 430.1220, Y 26.6154, Z -5.5000, A 0.000, B 0.000, C 0.000 }
gfCNCPoint4[15545] = {X 429.6706, Y 25.1508, Z -5.5000, A 0.000, B 0.000, C 0.000 }
gfCNCPoint4[15546] = {X 429.3565, Y 23.4677, Z -5.5000, A 0.000, B 0.000, C 0.000 }
gfCNCPoint4[15547] = {X 429.2162, Y 21.7614, Z -5.5000, A 0.000, B 0.000, C 0.000 }
gfCNCPoint4[15548] = {X 429.2509, Y 20.0497, Z -5.5000, A 0.000, B 0.000, C 0.000 }
gfCNCPoint4[15549] = {X 429.4603, Y 18.3505, Z -5.5000, A 0.000, B 0.000, C 0.000 }
gfCNCPoint4[15550] = {X 429.8423, Y 16.6816, Z -5.5000, A 0.000, B 0.000, C 0.000 }
gfCNCPoint4[15551] = {X 430.4014, Y 15.1284, Z -5.5000, A 0.000, B 0.000, C 0.000 }
gfCNCPoint4[15552] = {X 431.1711, Y 13.6683, Z -5.5000, A 0.000, B 0.000, C 0.000 }
gfCNCPoint4[15553] = {X 432.1367, Y 12.3295, Z -5.5000, A 0.000, B 0.000, C 0.000 }
gfCNCPoint4[15554] = {X 433.2792, Y 11.1381, Z -5.5000, A 0.000, B 0.000, C 0.000 }
gfCNCPoint4[15555] = {X 434.5764, Y 10.1174, Z -5.5000, A 0.000, B 0.000, C 0.000 }
gfCNCPoint4[15556] = {X 436.0030, Y 9.2871, Z -5.5000, A 0.000, B 0.000, C 0.000 }
gfCNCPoint4[15557] = {X 437.5314, Y 8.6636, Z -5.5000, A 0.000, B 0.000, C 0.000 }
gfCNCPoint4[15558] = {X 439.1317, Y 8.2588, Z -5.5000, A 0.000, B 0.000, C 0.000 }
gfCNCPoint4[15559] = {X 441.2287, Y 7.9685, Z -5.5000, A 0.000, B 0.000, C 0.000 }
gfCNCPoint4[15560] = {X 443.3436, Y 7.8743, Z -5.5000, A 0.000, B 0.000, C 0.000 }
gfCNCPoint4[15561] = {X 444.0357, Y 7.8702, Z -5.5000, A 0.000, B 0.000, C 0.000 }
gfCNCPoint4[15562] = {X 459.4468, Y 7.8702, Z -5.5000, A 0.000, B 0.000, C 0.000 }
gfCNCPoint4[15563] = {X 460.4061, Y 7.9783, Z -5.5000, A 0.000, B 0.000, C 0.000 }
gfCNCPoint4[15564] = {X 461.3173, Y 8.2972, Z -5.5000, A 0.000, B 0.000, C 0.000 }
gfCNCPoint4[15565] = {X 462.1347, Y 8.8108, Z -5.5000, A 0.000, B 0.000, C 0.000 }
gfCNCPoint4[15566] = {X 462.8174, Y 9.4934, Z -5.5000, A 0.000, B 0.000, C 0.000 }
gfCNCPoint4[15567] = {X 463.3310, Y 10.3109, Z -5.5000, A 0.000, B 0.000, C 0.000 }
gfCNCPoint4[15568] = {X 463.6499, Y 11.2221, Z -5.5000, A 0.000, B 0.000, C 0.000 }
gfCNCPoint4[15569] = {X 463.7579, Y 12.1814, Z -5.5000, A 0.000, B 0.000, C 0.000 }
gfCNCPoint4[15570] = {X 463.7579, Y 12.9782, Z -5.5000, A 0.000, B 0.000, C 0.000 }
gfCNCPoint4[15571] = {X 463.6566, Y 13.9079, Z -5.5000, A 0.000, B 0.000, C 0.000 }
gfCNCPoint4[15572] = {X 463.3575, Y 14.7940, Z -5.5000, A 0.000, B 0.000, C 0.000 }
gfCNCPoint4[15573] = {X 462.8748, Y 15.5950, Z -5.5000, A 0.000, B 0.000, C 0.000 }
gfCNCPoint4[15574] = {X 462.2309, Y 16.2733, Z -5.5000, A 0.000, B 0.000, C 0.000 }
gfCNCPoint4[15575] = {X 462.2311, Y 28.5935, Z -5.5000, A 0.000, B 0.000, C 0.000 }
gfCNCPoint4[15576] = {X 466.2311, Y 28.5934, Z -5.5000, A 0.000, B 0.000, C 0.000 }
gfCNCPoint4[15577] = {X 462.1511, Y 28.5935, Z -5.5000, A 0.000, B 0.000, C 0.000 }
gfCNCPoint4[15578] = {X 462.1514, Y 40.9516, Z -5.5000, A 0.000, B 0.000, C 0.000 }
gfCNCPoint4[15579] = {X 462.1885, Y 40.9821, Z -5.5000, A 0.000, B 0.000, C 0.000 }
gfCNCPoint4[15580] = {X 462.8113, Y 41.6401, Z -5.5000, A 0.000, B 0.000, C 0.000 }
gfCNCPoint4[15581] = {X 463.2800, Y 42.4154, Z -5.5000, A 0.000, B 0.000, C 0.000 }
gfCNCPoint4[15582] = {X 463.5733, Y 43.2725, Z -5.5000, A 0.000, B 0.000, C 0.000 }
gfCNCPoint4[15583] = {X 463.6778, Y 44.1724, Z -5.5000, A 0.000, B 0.000, C 0.000 }
gfCNCPoint4[15584] = {X 463.6779, Y 45.0000, Z -5.5000, A 0.000, B 0.000, C 0.000 }
gfCNCPoint4[15585] = {X 463.5716, Y 45.9435, Z -5.5000, A 0.000, B 0.000, C 0.000 }
gfCNCPoint4[15586] = {X 463.2580, Y 46.8397, Z -5.5000, A 0.000, B 0.000, C 0.000 }
gfCNCPoint4[15587] = {X 462.7529, Y 47.6436, Z -5.5000, A 0.000, B 0.000, C 0.000 }
gfCNCPoint4[15588] = {X 462.0815, Y 48.3150, Z -5.5000, A 0.000, B 0.000, C 0.000 }
gfCNCPoint4[15589] = {X 461.2776, Y 48.8201, Z -5.5000, A 0.000, B 0.000, C 0.000 }
gfCNCPoint4[15590] = {X 460.3814, Y 49.1337, Z -5.5000, A 0.000, B 0.000, C 0.000 }
gfCNCPoint4[15591] = {X 459.4379, Y 49.2400, Z -5.5000, A 0.000, B 0.000, C 0.000 }
gfCNCPoint4[15592] = {X 452.9945, Y 49.2400, Z -5.5000, A 0.000, B 0.000, C 0.000 }
gfCNCPoint4[15593] = {X 452.0558, Y 49.1348, Z -5.5000, A 0.000, B 0.000, C 0.000 }
gfCNCPoint4[15594] = {X 451.1636, Y 48.8243, Z -5.5000, A 0.000, B 0.000, C 0.000 }
gfCNCPoint4[15595] = {X 450.3624, Y 48.3241, Z -5.5000, A 0.000, B 0.000, C 0.000 }
gfCNCPoint4[15596] = {X 449.6918, Y 47.6589, Z -5.5000, A 0.000, B 0.000, C 0.000 }
gfCNCPoint4[15597] = {X 449.1851, Y 46.8617, Z -5.5000, A 0.000, B 0.000, C 0.000 }
gfCNCPoint4[15598] = {X 448.8674, Y 45.9721, Z -5.5000, A 0.000, B 0.000, C 0.000 }
gfCNCPoint4[15599] = {X 448.7546, Y 45.0343, Z -5.5000, A 0.000, B 0.000, C 0.000 }
gfCNCPoint4[15600] = {X 448.7549, Y 44.1505, Z -5.5000, A 0.000, B 0.000, C 0.000 }
gfCNCPoint4[15601] = {X 448.8654, Y 43.2454, Z -5.5000, A 0.000, B 0.000, C 0.000 }
gfCNCPoint4[15602] = {X 449.1668, Y 42.3850, Z -5.5000, A 0.000, B 0.000, C 0.000 }
gfCNCPoint4[15603] = {X 449.6452, Y 41.6088, Z -5.5000, A 0.000, B 0.000, C 0.000 }
gfCNCPoint4[15604] = {X 450.2784, Y 40.9529, Z -5.5000, A 0.000, B 0.000, C 0.000 }
gfCNCPoint4[15605] = {X 450.2784, Y 34.3938, Z -5.5000, A 0.000, B 0.000, C 0.000 }
gfCNCPoint4[15606] = {X 447.4261, Y 34.3938, Z -5.5000, A 0.000, B 0.000, C 0.000 }
gfCNCPoint4[15607] = {X 443.1027, Y 42.8116, Z -5.5000, A 0.000, B 0.000, C 0.000 }
gfCNCPoint4[15608] = {X 443.1192, Y 42.8570, Z -5.5000, A 0.000, B 0.000, C 0.000 }
gfCNCPoint4[15609] = {X 443.2817, Y 43.5053, Z -5.5000, A 0.000, B 0.000, C 0.000 }
gfCNCPoint4[15610] = {X 443.3403, Y 44.1710, Z -5.5000, A 0.000, B 0.000, C 0.000 }
gfCNCPoint4[15611] = {X 443.3405, Y 45.0000, Z -5.5000, A 0.000, B 0.000, C 0.000 }
gfCNCPoint4[15612] = {X 443.2342, Y 45.9435, Z -5.5000, A 0.000, B 0.000, C 0.000 }
gfCNCPoint4[15613] = {X 442.9206, Y 46.8397, Z -5.5000, A 0.000, B 0.000, C 0.000 }
gfCNCPoint4[15614] = {X 442.4154, Y 47.6436, Z -5.5000, A 0.000, B 0.000, C 0.000 }
gfCNCPoint4[15615] = {X 441.7441, Y 48.3150, Z -5.5000, A 0.000, B 0.000, C 0.000 }
gfCNCPoint4[15616] = {X 440.9401, Y 48.8201, Z -5.5000, A 0.000, B 0.000, C 0.000 }
gfCNCPoint4[15617] = {X 440.0440, Y 49.1337, Z -5.5000, A 0.000, B 0.000, C 0.000 }
gfCNCPoint4[15618] = {X 439.1005, Y 49.2400, Z -5.5000, A 0.000, B 0.000, C 0.000 }
gfCNCPoint4[15619] = {X 432.5144, Y 49.2400, Z -5.5000, A 0.000, B 0.000, C 0.000 }
gfCNCPoint4[15620] = {X 431.5709, Y 49.1337, Z -5.5000, A 0.000, B 0.000, C 0.000 }
gfCNCPoint4[15621] = {X 430.6748, Y 48.8201, Z -5.5000, A 0.000, B 0.000, C 0.000 }
gfCNCPoint4[15622] = {X 429.8708, Y 48.3150, Z -5.5000, A 0.000, B 0.000, C 0.000 }
gfCNCPoint4[15623] = {X 429.1995, Y 47.6436, Z -5.5000, A 0.000, B 0.000, C 0.000 }
gfCNCPoint4[15624] = {X 428.6943, Y 46.8397, Z -5.5000, A 0.000, B 0.000, C 0.000 }
gfCNCPoint4[15625] = {X 428.3807, Y 45.9436, Z -5.5000, A 0.000, B 0.000, C 0.000 }
gfCNCPoint4[15626] = {X 428.2744, Y 45.0001, Z -5.5000, A 0.000, B 0.000, C 0.000 }
gfCNCPoint4[15627] = {X 428.2748, Y 44.1505, Z -5.5000, A 0.000, B 0.000, C 0.000 }
gfCNCPoint4[15628] = {X 428.3718, Y 43.3054, Z -5.5000, A 0.000, B 0.000, C 0.000 }
gfCNCPoint4[15629] = {X 428.6354, Y 42.4967, Z -5.5000, A 0.000, B 0.000, C 0.000 }
gfCNCPoint4[15630] = {X 429.0552, Y 41.7570, Z -5.5000, A 0.000, B 0.000, C 0.000 }
gfCNCPoint4[15631] = {X 429.6142, Y 41.1158, Z -5.5000, A 0.000, B 0.000, C 0.000 }
gfCNCPoint4[15632] = {X 430.2899, Y 40.5992, Z -5.5000, A 0.000, B 0.000, C 0.000 }
gfCNCPoint4[15633] = {X 431.0551, Y 40.2278, Z -5.5000, A 0.000, B 0.000, C 0.000 }
gfCNCPoint4[15634] = {X 435.0928, Y 32.3244, Z -5.5000, A 0.000, B 0.000, C 0.000 }
gfCNCPoint4[15635] = {X 433.8198, Y 31.4679, Z -5.5000, A 0.000, B 0.000, C 0.000 }
gfCNCPoint4[15636] = {X 432.6744, Y 30.4470, Z -5.5000, A 0.000, B 0.000, C 0.000 }
gfCNCPoint4[15637] = {X 431.6777, Y 29.2804, Z -5.5000, A 0.000, B 0.000, C 0.000 }
gfCNCPoint4[15638] = {X 430.8482, Y 27.9895, Z -5.5000, A 0.000, B 0.000, C 0.000 }
gfCNCPoint4[15639] = {X 430.2011, Y 26.5983, Z -5.5000, A 0.000, B 0.000, C 0.000 }
gfCNCPoint4[15640] = {X 429.7484, Y 25.1323, Z -5.5000, A 0.000, B 0.000, C 0.000 }
gfCNCPoint4[15641] = {X 429.4358, Y 23.4572, Z -5.5000, A 0.000, B 0.000, C 0.000 }
gfCNCPoint4[15642] = {X 429.2961, Y 21.7590, Z -5.5000, A 0.000, B 0.000, C 0.000 }
gfCNCPoint4[15643] = {X 429.3307, Y 20.0554, Z -5.5000, A 0.000, B 0.000, C 0.000 }
gfCNCPoint4[15644] = {X 429.5391, Y 18.3643, Z -5.5000, A 0.000, B 0.000, C 0.000 }
gfCNCPoint4[15645] = {X 429.9193, Y 16.7033, Z -5.5000, A 0.000, B 0.000, C 0.000 }
gfCNCPoint4[15646] = {X 430.4746, Y 15.1607, Z -5.5000, A 0.000, B 0.000, C 0.000 }
gfCNCPoint4[15647] = {X 431.2392, Y 13.7104, Z -5.5000, A 0.000, B 0.000, C 0.000 }
gfCNCPoint4[15648] = {X 432.1982, Y 12.3806, Z -5.5000, A 0.000, B 0.000, C 0.000 }
gfCNCPoint4[15649] = {X 433.3330, Y 11.1973, Z -5.5000, A 0.000, B 0.000, C 0.000 }
gfCNCPoint4[15650] = {X 434.6215, Y 10.1834, Z -5.5000, A 0.000, B 0.000, C 0.000 }
gfCNCPoint4[15651] = {X 436.0385, Y 9.3588, Z -5.5000, A 0.000, B 0.000, C 0.000 }
